// TwinCAT 3 PLC project PShell_SampleTests
// ProgramVersion: 3.1.4023.0
// libraries:
//   CmpBitmapPool, * (System)
//   PShEll Universal Blocks, * (Precision Systems Engineering)
//   Tc2_MC2, * (Beckhoff Automation GmbH)
//   Tc2_Standard, * (Beckhoff Automation GmbH)
//   Tc2_System, * (Beckhoff Automation GmbH)
//   Tc2_TcpIp, * (Beckhoff Automation GmbH)
//   Tc3_EventLogger, * (Beckhoff Automation GmbH)
//   Tc3_McCollisionAvoidance, * (Beckhoff Automation GmbH)
//   Tc3_McCoordinatedMotion, * (Beckhoff Automation GmbH)
//   Tc3_Module, * (Beckhoff Automation GmbH)
//   VisuDialogs, * (System)
//   VisuSymbols,3.5.10.0,System
// project tree:
//   DUTs/Fixture/ E_FcqFixtureStateGSampleMeas.TcDUT, E_FixtureJigStateAbort.TcDUT, E_FixtureJigStateInit.TcDUT, E_FixtureJigStateReset.TcDUT, E_FixtureLoadNormResult.TcDUT, E_FixtureMeasurementResultExt.TcDUT, E_FixtureState.TcDUT, E_FixtureStateAbort.TcDUT, E_FixtureStateInit.TcDUT, E_FixtureStateLoadNorm.TcDUT, E_FixtureStateMeasurement.TcDUT, E_FixtureStateMeasurementDataExchange.TcDUT, E_FixtureStateReset.TcDUT, E_FixtureStateTest.TcDUT, E_GoldenSampleState.TcDUT
//   DUTs/ ST_Shell.TcDUT, ST_ShellFlags.TcDUT, ST_ShellPlatform.TcDUT, ST_ShellRecipeData.TcDUT
//   / GlobalTextList.TcGTLO, RecipeManager.TcRMO (not stored), SampleTests.TcTTO, VisualizationManager.TcVMO (not stored), VISU_TASK.TcTTO
//   GVLs/ GVL.TcGVL
//   POUs/Platform Tests/Alarm Control/ PRG_AlarmControl.TcPOU
//   POUs/Platform Tests/Machine Control/ FB_MachineControl.TcPOU, I_MachineControl.TcIO, PRG_MachineControl.TcPOU
//   POUs/Platform Tests/Visu Control/ FB_VisuControl.TcPOU, F_CloseDialog.TcPOU, F_OpenDialog.TcPOU, PRG_VisuControl.TcPOU
//   POUs/Platform Tests/Recipes Manager/ PRG_RecipesManager.TcPOU
//   POUs/Universal Blocks/Alarms/ PRG_FB_AlarmControler_Test.TcPOU
//   POUs/Universal Blocks/Analog Devices/Analog Input/ PRG_FB_AnalogInput_Test.TcPOU
//   POUs/Universal Blocks/Analog Devices/Analog Output/ PRG_FB_AnalogOutput_Test.TcPOU
//   POUs/Universal Blocks/Axis CA/ PRG_FB_AxisServoCA_PreTest.TcPOU, PRG_FB_AxisServoCA_Test.TcPOU, PRG_FB_MoverCA_Test.TcPOU, PRG_FB_Axis_JennyScienceEthCA_Test.TcPOU
//   POUs/Universal Blocks/Axis/ PRG_FB_Axis_Faulhaber_Test.TcPOU (excluded from build), PRG_FB_Axis_JennyScienceEthSingle_Test.TcPOU (excluded from build), PRG_FB_AxisServo_Test.TcPOU
//   POUs/Universal Blocks/Communication/Backhoff ADS/ PRG_FB_AdsExchanger_Test.TcPOU
//   POUs/Universal Blocks/Communication/TcpIp/ PRG_FB_TcpClient_Test.TcPOU, PRG_FB_TcpServer_Test.TcPOU, PRG_FUN_TcpDataConversion_Test.TcPOU
//   POUs/Universal Blocks/Cylinder/ PRG_FB_SingleCoilCylinder_Test.TcPOU, PRG_FB_DoubleCoilCylinder_Test.TcPOU
//   POUs/Universal Blocks/Digital Devices/Beacon/ PRG_FB_Beacon_Test.TcPOU
//   POUs/Universal Blocks/Digital Devices/Digital Input/ PRG_FB_DigitalInput_Test.TcPOU, PRG_FB_DigitalInputExt_Test.TcPOU
//   POUs/Universal Blocks/Digital Devices/Digital Output/ PRG_FB_DigitalOutput_Test.TcPOU
//   POUs/Universal Blocks/Digital Devices/Lamp/ PRG_FB_Lamp_Test.TcPOU
//   POUs/Universal Blocks/Fixtures/ FB_Fixture222.TcPOU, PRG_FB_FixtureCommTest.TcPOU
//   POUs/Universal Blocks/Fixture/ FB_FixtureClamp.TcPOU, FB_FixtureJig.TcPOU, FB_Fixture.TcPOU, PRG_FB_FcqFixture_Development_Test.TcPOU
//   POUs/Universal Blocks/Robots/ PRG_FB_CR800.TcPOU
//   POUs/Universal Blocks/Utilities/Beckhoff UPS/ PRG_FB_UpsCx20xx_Test.TcPOU, PRG_FB_UpsCx50xx_Test.TcPOU
//   POUs/Universal Blocks/Utilities/CSV Data Exchanger/ PRG_FB_CSVDataExchanger_Test.TcPOU
//   POUs/Universal Blocks/Utilities/File Logger/ PRG_FB_FileLogger_Test.TcPOU
//   POUs/Universal Blocks/Utilities/Recipes Manager/ PRG_FB_RecipesManager_Test.TcPOU
//   POUs/Universal Blocks/Utilities/StringMerge/ PRG_FUN_MergeStringsX_Test.TcPOU
//   POUs/Universal Blocks/Utilities/TXT Data Exchanger/ PRG_FB_TXTDataExchanger_Test.TcPOU
//   POUs/Universal Blocks/Vision/ PRG_FB_Camera_Test.TcPOU
//   POUs/Universal Blocks/XTS/ FB_XtsStation.TcPOU, PRG_XtsControlUnit_Test.TcPOU
//   VISUs/Platform/Pages/ PageAuto.TcVIS, PageInitializing.TcVIS, PageManualOther.TcVIS, PageUninitialized.TcVIS
//   VISUs/Platform/ ShellMainVisu.TcVIS

CONFIGURATION PShell_SampleTests
    RESOURCE PLC ON TwinCAT3
        TASK SampleTests(INTERVAL := T#10ms, PRIORITY := 20);
        TASK VISU_TASK(INTERVAL := T#200000us, PRIORITY := 30);
        PROGRAM PRG_MachineControl WITH SampleTests : PRG_MachineControl;
        PROGRAM PRG_AlarmControl WITH SampleTests : PRG_AlarmControl;
        PROGRAM PRG_RecipesManager WITH SampleTests : PRG_RecipesManager;
        PROGRAM PRG_VisuControl WITH SampleTests : PRG_VisuControl;
        PROGRAM VisuElems_Visu_Prg WITH VISU_TASK : VisuElems.Visu_Prg;
    END_RESOURCE
END_CONFIGURATION

// ---- DUTs/Fixture/E_FcqFixtureStateGSampleMeas.TcDUT

{attribute 'strict'}
TYPE E_FcqFixtureStateGSampleMeas :
(
	FIXTURE_GOLDEN_SAMPLE_CLOSE								:= 0,
	FIXTURE_GOLDEN_SAMPLE_SEND_MEASURE_COMMAND				:= 10,
	FIXTURE_GOLDEN_SAMPLE_WAIT_FOR_RESPONSE 				:= 20,
	FIXTURE_GOLDEN_SAMPLE_OPEN								:= 30,
	FIXTURE_GOLDEN_SAMPLE_MEASUREMENT_DONE					:= 40,
	FIXTURE_GOLDEN_SAMPLE_WAIT_FOR_UTU						:= 50
	
	
);
END_TYPE

// ---- DUTs/Fixture/E_FixtureJigStateAbort.TcDUT
{attribute 'strict'}
TYPE E_FixtureJigStateAbort :
(
	FIXTURE_JIG_ABORT_JIG_PUSHER	:= 0,	(*  *)
	FIXTURE_JIG_ABORT_DONE			:= 10	(*  *)
);
END_TYPE

// ---- DUTs/Fixture/E_FixtureJigStateInit.TcDUT
{attribute 'strict'}
TYPE E_FixtureJigStateInit :
(
	FIXTURE_JIG_INIT_JIG_PUSHER	:= 0,	(*  *)
	FIXTURE_JIG_INIT_DONE		:= 10	(*  *)
);
END_TYPE

// ---- DUTs/Fixture/E_FixtureJigStateReset.TcDUT
{attribute 'strict'}
TYPE E_FixtureJigStateReset :
(
	FIXTURE_JIG_RESET_JIG_PUSHER	:= 10,	(*  *)
	FIXTURE_JIG_RESET_DONE			:= 0	(*  *)
);
END_TYPE

// ---- DUTs/Fixture/E_FixtureLoadNormResult.TcDUT
{attribute 'strict'}
TYPE E_FixtureLoadNormResult :
(
	FIXTURE_NORM_LOAD_UNKNOWN				:= 0,	(*  *)
	FIXTURE_NORM_LOAD_SUCCESS				:= 10,	(*  *)
	FIXTURE_NORM_LOAD_FAIL					:= 20,	(*  *)
	FIXTURE_NORM_LOAD_GOLDEN_SAMPLE_NEEDED 	:= 30	(*	*)
);
END_TYPE

// ---- DUTs/Fixture/E_FixtureMeasurementResultExt.TcDUT
{attribute 'strict'}
TYPE E_FixtureMeasurementResultExt :
(
	FIXTURE_MEASUREMENT_RESULT_NONE			:= 0,
	FIXTURE_MEASUREMENT_RESULT_GOOD			:= 10,
	FIXTURE_MEASUREMENT_RESULT_THD 			:= 20,
	FIXTURE_MEASUREMENT_RESULT_PHASE		:= 30,
	FIXTURE_MEASUREMENT_RESULT_SSPL			:= 40,
	FIXTURE_MEASUREMENT_RESULT_RUBBING		:= 50,
	FIXTURE_MEASUREMENT_RESULT_IMP			:= 60,
	FIXTURE_MEASUREMENT_RESULT_HFA			:= 70,
	FIXTURE_MEASUREMENT_RESULT_SPL			:= 80,
	FIXTURE_MEASUREMENT_RESULT_CONNECT		:= 90,
	FIXTURE_MEASUREMENT_RESULT_REJECT_OTHER	:= 100,
	FIXTURE_MEASUREMENT_RESULT_REWORK		:= 110
);
END_TYPE

// ---- DUTs/Fixture/E_FixtureState.TcDUT
{attribute 'strict'}
TYPE E_FixtureState :
(
	FIXTURE_EXTENSION_IDLE								:= 0,	(*  *)
	FIXTURE_EXTENSION_COVER_ACTIVE	 					:= 10,	(*  *)
	FIXTURE_EXTENSION_COVER_ACTIVE_DONE					:= 20,	(*  *)
	FIXTURE_EXTENSION_COVER_HOME						:= 30,	(*  *)
	FIXTURE_EXTENSION_COVER_HOME_DONE					:= 40,	(*  *)
	FIXTURE_EXTENSION_CLAMP_HOLD						:= 50,	(*  *)
	FIXTURE_EXTENSION_CLAMP_HOLD_DONE					:= 60,	(*  *)
	FIXTURE_EXTENSION_CLAMP_RELEASE						:= 70,	(*  *)
	FIXTURE_EXTENSION_CLAMP_RELEASE_DONE				:= 80,	(*  *)
	FIXTURE_EXTENSION_COVER_ACTIVE_AND_JIG_OPEN			:= 90,	(*  *)
	FIXTURE_EXTENSION_COVER_ACTIVE_AND_JIG_OPEN_DONE 	:= 100,	(*  *)
	FIXTURE_EXTENSION_COVER_HOME_AND_JIG_CLOSE			:= 110,	(*  *)
	FIXTURE_EXTENSION_COVER_HOME_AND_JIG_CLOSE_DONE		:= 120,	(*  *)
	FIXTURE_EXTENSION_LOAD_NORM							:= 130,	(*  *)
	FIXTURE_EXTENSION_LOAD_NORM_DONE					:= 140,	(*  *)
	FIXTURE_EXTENSION_GOLDEN_SAMPLE_MEASURE				:= 150,	(*	*)
	FIXTURE_EXTENSION_GOLDEN_SAMPLE_MEASURE_DONE		:= 160	(*  *)
);
END_TYPE

// ---- DUTs/Fixture/E_FixtureStateAbort.TcDUT
{attribute 'strict'}
TYPE E_FixtureStateAbort :
(
	FIXTURE_ABORT_CLAMP		:= 0,	(*  *)
	FIXTURE_ABORT_COVER		:= 20,	(*  *)
	FIXTURE_ABORT_DONE	:= 10	(*  *)
);
END_TYPE

// ---- DUTs/Fixture/E_FixtureStateInit.TcDUT
{attribute 'strict'}
TYPE E_FixtureStateInit :
(
	FIXTURE_INIT_CLAMP	:= 0,	(*  *)
	FIXTURE_INIT_COVER	:= 20,	(*  *)
	FIXTURE_INIT_DONE	:= 10	(*  *)
);
END_TYPE

// ---- DUTs/Fixture/E_FixtureStateLoadNorm.TcDUT
{attribute 'strict'}
TYPE E_FixtureStateLoadNorm :
(
	FIXTURE_LOADING_NORM_SEND_NORM_DATA 				:= 0,	(*  *)
	FIXTURE_LOADING_NORM_WAIT_FOR_RESPONSE				:= 10,	(*  *)
	FIXTURE_LOADING_NORM_DONE							:= 20,	(*  *)
	FIXTURE_LOADING_NORM_GOLDEN_SAMPLE_TEST 			:= 30,	(*	*)
	FIXTURE_LOADING_NORM_GOLDEN_SAMPLE_WAIT_FOR_END		:= 40	(*	*)
);
END_TYPE

// ---- DUTs/Fixture/E_FixtureStateMeasurement.TcDUT
{attribute 'strict'}
TYPE E_FixtureStateMeasurement :
(
	FIXTURE_MEASUREMENT_START 				:= 0,
	FIXTURE_MEASUREMENT_WAIT_FOR_BUSY 		:= 10,
	FIXTURE_MEASUREMENT_WAIT_FOR_RESPONSE 	:= 20,
	FIXTURE_MEASUREMENT_REMEASUREMENT		:= 30,
	FIXTURE_MEASUREMENT_DONE				:= 40
);
END_TYPE

// ---- DUTs/Fixture/E_FixtureStateMeasurementDataExchange.TcDUT
{attribute 'strict'}
TYPE E_FixtureStateMeasurementDataExchange :
(
	FIXTURE_MEASURE_DATA_EXCHANGING_WAIT_FOR_BUSY 		:= 0,
	FIXTURE_MEASURE_DATA_EXCHANGING_WAIT_FOR_FISNISH 	:= 10,
	FIXTURE_MEASURE_DATA_EXCHANGING_PROCCESS_RESULTS 	:= 20,
	FIXTURE_MEASURE_DATA_EXCHANGING_DONE				:= 30
);
END_TYPE

// ---- DUTs/Fixture/E_FixtureStateReset.TcDUT
{attribute 'strict'}
TYPE E_FixtureStateReset :
(
	FIXTURE_RESET_CLAMP	:= 0,	(*  *)
	FIXTURE_RESET_COVER	:= 10,	(*  *)
	FIXTURE_RESET_DONE	:= 20	(*  *)
);
END_TYPE

// ---- DUTs/Fixture/E_FixtureStateTest.TcDUT
{attribute 'strict'}
TYPE E_FixtureStateTest :
(
	FIXTURE_TEST_WAIT_FOR_COMMAND 			:= 0,	(*  *)
	FIXTURE_TEST_INIT						:= 10,	(*  *)
	FIXTURE_TEST_OPEN						:= 20,	(*  *)
	FIXTURE_TEST_CLOSE						:= 30,	(*  *)
	FIXTURE_TEST_MEASURE					:= 40,	(*  *)
	FIXTURE_TEST_RESET						:= 50,	(*  *)
	FIXTURE_TEST_PLATFORM_HOME				:= 60,	(*  *)
	FIXTURE_TEST_PLATFORM_ACTIVE			:= 70,	(*  *)
	FIXTURE_TEST_PRODUCT_HOLD				:= 80,	(*  *)
	FIXTURE_TEST_PRODUCT_RELEASE			:= 90,	(*  *)
	FIXTURE_TEST_PLATFORM_ACTIVE_AND_OPEN	:= 100,	(*  *)
	FIXTURE_TEST_PLATFORM_HOME_AND_CLOSE	:= 110,	(*  *)
	FIXTURE_TEST_LOAD_NORM					:= 120,	(*  *)
	FIXTURE_TEST_MEASUREMENT				:= 130,	(*  *)
	FIXTURE_START_POS						:= 210,
	FIXTURE_TEST_HOME						:= 220,
	FIXTURE_TEST_ERROR						:= 999,
	FIXTURE_TEST_ABORT						:= -10	(*  *)
);
END_TYPE

// ---- DUTs/Fixture/E_GoldenSampleState.TcDUT
{attribute 'strict'}
TYPE E_GoldenSampleState :
(
	GS_STATUS_UNKNOWN		:= 0,
	GS_STATUS_BCHECKSETUP	:= 10,
	GS_STATUS_NOK			:= 20,
	GS_STATUS_OK			:= 30
);
END_TYPE

// ---- DUTs/ST_Shell.TcDUT
TYPE ST_Shell :
STRUCT
	stPlatform		: ST_ShellPlatform;		(*  *)
	stFlags			: ST_ShellFlags;		(*  *)
	stRecipeData	: ST_ShellRecipeData;	(*  *)
END_STRUCT
END_TYPE

// ---- DUTs/ST_ShellFlags.TcDUT
TYPE ST_ShellFlags :
STRUCT
	bMachineCtrlAssignamentsDone	: BOOL := FALSE;	(*  *)
	bVisuCtrlAssignamentsDone		: BOOL := FALSE;	(*  *)
	bAlarmCtrlAssignamentsDone		: BOOL := FALSE;	(*  *)
	bRecipesCtrlAssignamentsDone	: BOOL := FALSE;	(*  *)
END_STRUCT
END_TYPE

// ---- DUTs/ST_ShellPlatform.TcDUT
TYPE ST_ShellPlatform EXTENDS ST_UniversalPlatform :
STRUCT
	ref_fbMachineControler : REFERENCE TO FB_MachineControl;	(*  *)
	//refFbMachineSafety	: REFERENCE TO FB_MachineSafety;	(*  *)
	ref_fbVisuControler	: REFERENCE TO FB_VisuControl;			(*  *)
END_STRUCT
END_TYPE

// ---- DUTs/ST_ShellRecipeData.TcDUT
TYPE ST_ShellRecipeData :
STRUCT
	(* Add recipe variables here and link them with RecipeManager in Tc3 XAE Shell *)
	rpVar1 : FB_RecipeParameter;
	rpVar2 : FB_RecipeParameter;
	rpVar3 : FB_RecipeParameter;
	rpVar4 : FB_RecipeParameter;
	rpVar5 : FB_RecipeParameter;
	rpVar6 : FB_RecipeParameter;
	rpVar7 : FB_RecipeParameter;
	rpVar8 : FB_RecipeParameter;
	rpVar9 : FB_RecipeParameter;
    rpVar10 : FB_RecipeParameter;
END_STRUCT
END_TYPE

// ---- GVLs/GVL.TcGVL
VAR_GLOBAL
	stShell : ST_Shell;	(* This structure contains references to Shell modules, recipe parameters and auxilary bit flags *)

	(* Measurement FCQ fixtures *)
	sFIXTURE_NAME								: STRING		:= 'Fixture';
	sFIXTURE_HOST								: T_IPv4Addr	:= '192.168.0.';
	sFIXTURE_AMS_NET_ID							: T_AmsNetID	:= '';
	iFIXTURE_PORT								: UINT			:= 400;
	tFIXTURE_TIMEOUT							: TIME			:= DEFAULT_ADS_TIMEOUT;
	bFIXTURE_USE_LOGGER							: BOOL			:= FALSE;
	bFIXTURE_USE_CLIENT							: BOOL			:= TRUE;
	sFIXTURE_LOGGER_NAME						: STRING		:= 'Logger_Fixture_';
	sFIXTURE_FILE_DIR							: STRING		:= 'C:\Fixture_';
END_VAR

// ---- POUs/Platform Tests/Machine Control/I_MachineControl.TcIO
INTERFACE I_MachineControl EXTENDS I_UniversalMachine

PROPERTY Axes : REFERENCE TO ARRAY[0..19] OF FB_AxisServo
GET
END_GET
END_PROPERTY

PROPERTY DoubleCoilCylinders : REFERENCE TO ARRAY[0..9] OF FB_DoubleCoilCylinder
GET
END_GET
END_PROPERTY

PROPERTY Inputs : REFERENCE TO ARRAY[0..19] OF FB_DigitalInput
GET
END_GET
END_PROPERTY

PROPERTY Outputs : REFERENCE TO ARRAY[0..19] OF FB_DigitalOutput
GET
END_GET
END_PROPERTY

PROPERTY Robots : REFERENCE TO ARRAY[0..9] OF  FB_CR800EtherCAT
GET
END_GET
END_PROPERTY

PROPERTY SafeInputs : REFERENCE TO ARRAY[0..19] OF FB_DigitalInput
GET
END_GET
END_PROPERTY

PROPERTY SafeOutputs : REFERENCE TO ARRAY[0..19] OF FB_DigitalOutput
GET
END_GET
END_PROPERTY

PROPERTY SingleCoilCylinders : REFERENCE TO ARRAY[0..9] OF FB_SingleCoilCylinder
GET
END_GET
END_PROPERTY

END_INTERFACE

// ---- POUs/Platform Tests/Machine Control/PRG_MachineControl.TcPOU
PROGRAM PRG_MachineControl
VAR
	bFirstCycle 		: BOOL := TRUE;			(*  *)
	fbMachineControler 	: FB_MachineControl;	(*  *)
	fbFileLogger 		: FB_FileLogger;		(*	*)
END_VAR

IF bFirstCycle THEN
	bFirstCycle := FALSE;
	
	(* Assign machine controler reference to Shell API*)
	stShell.stPlatform.ref_fbMachineControler REF= fbMachineControler;
	
	(* Set assignamnet done bit for visu controler *)
	stShell.stFlags.bMachineCtrlAssignamentsDone := TRUE;
	
	fbMachineLogger.MR_FirstCycle( 	sName		:= 'PSE_Shell_Machine_Logger',
									sFileDir 	:= 'C:\TwinCAT\Projects\Loggers',
									sFileName 	:= 'PSE_Shell_Machine_Logger',
									sAmsNetId 	:= '',
									bAddTimeStamp := FALSE,
									bAddHeader := FALSE);
END_IF

IF NOT fbMachineLogger.Active THEN 
	fbMachineLogger.MR_Init();	
END_IF

fbMachineTime(bEnable := TRUE);
fbMachineControler();
fbMachineLogger();

END_PROGRAM

// ---- POUs/Platform Tests/Machine Control/FB_MachineControl.TcPOU
FUNCTION_BLOCK FB_MachineControl EXTENDS FB_UniversalMachine IMPLEMENTS I_MachineControl
VAR
	iLoop : USINT;	(* for loop auxilary variable *)

	(* --- Sample actuators - from shell template --- DELETE IF NOT NEEDED - *)
	arrDigitalInput		: ARRAY[0..19] OF FB_DigitalInput;			(* Array of sample digital inputs *)
	arrDigitalOutput	: ARRAY[0..19] OF FB_DigitalOutput;			(* Array of sample digital outputs *)
	arrCylinderDc		: ARRAY[0..9] OF FB_DoubleCoilCylinder;		(* Array of sample double coil cylinders *)
	arrCylinderSc		: ARRAY[0..9] OF FB_SingleCoilCylinder;		(* Array of sample single coil cylinders *)
	arrAxis				: ARRAY[0..19] OF FB_AxisServo;				(* Array of sample axis *)
	arrRobot			: ARRAY[0..9] OF FB_CR800EtherCAT;			(* Array of sample robots *)
	
	tonTestDelay	: TON;	(* Delay which allows to see any page changes during tests *)
	(* --- Sample actuators - from shell template --- DELETE IF NOT NEEDED - *)
	
	bStart			: BOOL;
	
	(* CR800 - testing *)
	lrPositionX1 : LREAL := 203.733;
	lrPositionY1 : LREAL := 100.000;
	lrRotation1  : LREAL := 216.699;
	
	lrPositionX2 : LREAL := -13.733;
	lrPositionY2 : LREAL := 8.001;
	lrRotation2  : LREAL := -2.889;
	
	
	bUserDefinedArea1	: BOOL;
	bTryIt1				: BOOL;
	bTryIt2				: BOOL;
END_VAR

IF bFirstCycle THEN
	(* bFirstCycle bit reset by parent *)
	(* --- Assign initial parameters for machine objects ---*)
	(* ---- DELETE IF NOT NEEDED ---- *)
	(* Assign sample digital inputs *)
	FOR iLoop := 0 TO 19 DO
		arrDigitalInput[iLoop].MR_FirstCycle(CONCAT('Digital_Input_',USINT_TO_STRING(iLoop)),CONCAT('EL1008-',USINT_TO_STRING(iLoop/8)),USINT_TO_STRING(iLoop MOD 8));
	END_FOR
	
	(* Assign sample digital outputs *)
	FOR iLoop := 0 TO 19 DO
		arrDigitalOutput[iLoop].MR_FirstCycle(CONCAT('Digital_Output_',USINT_TO_STRING(iLoop)),CONCAT('EL2008-',USINT_TO_STRING(iLoop/8)),USINT_TO_STRING(iLoop MOD 8));
	END_FOR
	
	(* Assign sample cylinders *)
	FOR iLoop := 0 TO 9 DO
		arrCylinderDc[iLoop].MR_FirstCycle(	sName					:= CONCAT('Double_Coil_Cylinder_',USINT_TO_STRING(iLoop)),
											sActiveSensorModuleType :=CONCAT('EL1008-',USINT_TO_STRING(iLoop/4)),
											sActiveSensorPortID 	:= USINT_TO_STRING(iLoop*2),
											sHomeSensorModuleType	:=CONCAT('EL1008-',USINT_TO_STRING(iLoop/4)),
											sHomeSensorPortID		:= USINT_TO_STRING(iLoop*2+1),
											tGoHomeTimeout			:= T#10S,
											tGoActiveTimeout		:= T#10S,
											tDelay 					:= T#1S);
		arrCylinderDc[iLoop].Simulation := TRUE;
		arrCylinderDc[iLoop].ref_poActiveValve.ModuleType := CONCAT('EL2008-',USINT_TO_STRING(iLoop/4));
		arrCylinderDc[iLoop].ref_poActiveValve.PortID := USINT_TO_STRING(iLoop*2);
		arrCylinderDc[iLoop].ref_poHomeValve.ModuleType := CONCAT('EL2008-',USINT_TO_STRING(iLoop/4));
		arrCylinderDc[iLoop].ref_poHomeValve.PortID := USINT_TO_STRING(iLoop*2+1);
	END_FOR
	
	FOR iLoop := 0 TO 9 DO
		arrCylinderSc[iLoop].MR_FirstCycle(	sName				:= CONCAT('Single_Coil_Cylinder_', USINT_TO_STRING(iLoop)),
											sActiveSensorModuleType :=CONCAT('EL1008-',USINT_TO_STRING(iLoop/4)),
											sActiveSensorPortID :=USINT_TO_STRING(iLoop*2),
											sHomeSensorModuleType :=CONCAT('EL1008-',USINT_TO_STRING(iLoop/4)),
											sHomeSensorPortID	:=USINT_TO_STRING(iLoop*2+1),
											tGoHomeTimeout 		:= T#12S,
											tGoActiveTimeout 	:= T#12S,
											tDelay 				:= T#2S);
		arrCylinderSc[iLoop].Simulation := TRUE;
		arrCylinderSc[iLoop].ref_poActiveValve.ModuleType := CONCAT('EL2008-',USINT_TO_STRING(iLoop/8));
		arrCylinderSc[iLoop].ref_poActiveValve.PortID := USINT_TO_STRING(iLoop);
	END_FOR
	
	(* Assign sample axes *)
	FOR iLoop := 0 TO 19 DO
		arrAxis[iLoop].MR_FirstCycle( 	sName 				:= CONCAT('Axis_',USINT_TO_STRING(iLoop)),
										sMeasurementUnits 	:= 'mm',
										bModulo				:= FALSE);
		arrAxis[iLoop].ref_HomeSwitch.ModuleType :=CONCAT('EL1008-',USINT_TO_STRING(iLoop/8));
		arrAxis[iLoop].ref_HomeSwitch.PortID :=USINT_TO_STRING(iLoop MOD 8);			
	END_FOR	
	
	(* Assign sample robots *)
	FOR iLoop := 0 TO 9 DO
		arrRobot[iLoop].MR_FirstCycle(	sName		:= CONCAT('Robot_',USINT_TO_STRING(iLoop)),
										iOverride	:= 100);
	END_FOR
	(* ---- DELETE IF NOT NEEDED ---- *)
END_IF

(* Execute parent implementation *)
SUPER^();

(* --- Cyclic run of internal objects ---*)
(* ---- DELETE IF NOT NEEDED ---- *)
(* Cyclic run of sample inputs *)
FOR iLoop := 0 TO 19 DO
	arrDigitalInput[iLoop]();
END_FOR

(* Cyclic run of sample outputs *)
FOR iLoop := 0 TO 19 DO
	arrDigitalOutput[iLoop]();
END_FOR
	
(* Cyclic run of sample double coil cylinders *)
FOR iLoop := 0 TO 9 DO
	arrCylinderDc[iLoop]();
END_FOR

(* Cyclic run of sample single coil cylinders *)
FOR iLoop := 0 TO 9 DO
	arrCylinderSc[iLoop]();
END_FOR

(* Cyclic run of sample axis *)
FOR iLoop := 0 TO 19 DO
	arrAxis[iLoop]();
END_FOR

(* Cyclic run of sample robots *)
FOR iLoop := 0 TO 9 DO
	arrRobot[iLoop]();
END_FOR

IF bTryIt1 THEN
	arrRobot[0].MR_SendPosition1( lrPositionX1 := lrPositionX1,
								lrPositionY1 := lrPositionY1,
								lrRotation1  := lrRotation1);
	IF NOT arrRobot[0].SendingPosition1 THEN
		bTryIt1 := FALSE;
	END_IF
END_IF

IF bTryIt2 THEN
	arrRobot[0].MR_SendPosition2( lrPositionX2 := lrPositionX2,
								lrPositionY2 := lrPositionY2,
								lrRotation2  := lrRotation2);
	IF NOT arrRobot[0].SendingPosition2 THEN
		bTryIt1 := FALSE;
	END_IF
END_IF

bUserDefinedArea1 := arrRobot[0].UserDefinedArea1;

tonTestDelay();
(* ---- DELETE IF NOT NEEDED ---- *)

PROPERTY Axes : REFERENCE TO ARRAY[0..19] OF FB_AxisServo
GET
Axes REF= arrAxis;
END_GET
END_PROPERTY

PROPERTY DoubleCoilCylinders : REFERENCE TO ARRAY[0..9] OF FB_DoubleCoilCylinder
GET
DoubleCoilCylinders REF= arrCylinderDc;
END_GET
END_PROPERTY

PROPERTY Inputs : REFERENCE TO ARRAY[0..19] OF FB_DigitalInput
GET
Inputs REF= arrDigitalInput;
END_GET
END_PROPERTY

METHOD MR_Start : BOOL
VAR_INPUT
END_VAR
bRunning := TRUE;

IF NOT bStart THEN
	fbMsgAutoStarted.Send(0);
	bStart := TRUE;
END_IF
END_METHOD

METHOD MR_Stop : BOOL
VAR_INPUT
END_VAR
bRunning := FALSE;

IF bStart THEN
	fbMsgAutoStopped.Send(0);
	bStart := FALSE;
END_IF
END_METHOD

METHOD PROTECTED MS_Aborting
VAR_INPUT
END_VAR
(* 
Add here code to abort all machine objects's e.g robots, axes, cylinders. 
At the end add "eMachineState := MACHINE_STATE_UNINITIALIZED;" to finish aborting.
*)
(* Aborting simulation - DELETE *)
tonTestDelay(IN := TRUE, PT:= T#4S);
IF tonTestDelay.Q THEN
	tonTestDelay(IN := FALSE);
	eMachineState := MACHINE_STATE_UNINITIALIZED;
END_IF
END_METHOD

METHOD PROTECTED MS_Auto
VAR_INPUT
END_VAR
(* 
Add here code to perform automatic process.
*)
;
END_METHOD

METHOD PROTECTED MS_AutoToManual
VAR_INPUT
END_VAR
(* 
Add here code to switch machine into manual mode. 
At the end add "eMachineState := MACHINE_STATE_MANUAL;" to finish switching.
*)
(* Switching mode to manual simulation - DELETE *)
tonTestDelay(IN := TRUE, PT:= T#4S);
bRunning := FALSE;
IF tonTestDelay.Q THEN
	tonTestDelay(IN := FALSE);
	eMachineState := MACHINE_STATE_MANUAL;
END_IF
END_METHOD

METHOD PROTECTED MS_Emergency
VAR_INPUT
END_VAR
END_METHOD

METHOD PROTECTED MS_Initializing
VAR_INPUT
END_VAR
(* 
Add here code to initialize all machine objects's e.g robots, axes, cylinders. 
At the end add "eMachineState := MACHINE_STATE_READY_INITIALIZED;" to finish initialization.
*)
(* Initialization simulation - DELETE  *)
tonTestDelay(IN := TRUE, PT:= T#4S);
IF tonTestDelay.Q THEN
	tonTestDelay(IN := FALSE);
	eMachineState := MACHINE_STATE_READY_INITIALIZED;
END_IF
END_METHOD

METHOD PROTECTED MS_Manual
VAR_INPUT
END_VAR
(* 
Leave empty - manual mode is provided by HMI controler and automatic frame generator.
*)
;
END_METHOD

METHOD PROTECTED MS_ManualToAuto
VAR_INPUT
END_VAR
(* 
Add here code to switch machine into auto mode. 
At the end add "eMachineState := MACHINE_STATE_MANUAL;" to finish switching.
*)
(* Switching mode to auto simulation - DELETE *)
tonTestDelay(IN := TRUE, PT:= T#4S);
IF tonTestDelay.Q THEN
	tonTestDelay(IN := FALSE);
	eMachineState := MACHINE_STATE_AUTO;
END_IF
END_METHOD

METHOD PROTECTED MS_ReadyInitialized
VAR_INPUT
END_VAR
(*
Add code here if some internal parameters are needed to set after initialization or leave it default.
At the end add "eMachineState := MACHINE_STATE_AUTO;" to finish and go to IDLE state.
*)
(* Ready-Initialized simulation - DELETE  *)
tonTestDelay(IN := TRUE, PT:= T#4S);
IF tonTestDelay.Q THEN
	tonTestDelay(IN := FALSE);
	eMachineState := MACHINE_STATE_AUTO;
END_IF
END_METHOD

METHOD PROTECTED MS_Reset
VAR_INPUT
END_VAR
(* 
Add here code to reset all machine objects's e.g robots, axes, cylinders. 
At the end add "eMachineState := MACHINE_STATE_RESET_DONE;" to finish reseting.
*)
(* Reset simulation - DELETE  *)
tonTestDelay(IN := TRUE, PT:= T#4S);
IF tonTestDelay.Q THEN
	tonTestDelay(IN := FALSE);
	eMachineState := MACHINE_STATE_RESET_DONE;
END_IF
END_METHOD

METHOD PROTECTED MS_ResetDone
VAR_INPUT
END_VAR
eMachineState := eMachineStateBeforeReset;
END_METHOD

METHOD PROTECTED MS_Uninitialized
VAR_INPUT
END_VAR
;
END_METHOD

PROPERTY Outputs : REFERENCE TO ARRAY[0..19] OF FB_DigitalOutput
GET
Outputs REF= arrDigitalOutput;
END_GET
END_PROPERTY

PROPERTY Robots : REFERENCE TO ARRAY[0..9] OF FB_CR800EtherCAT
GET
Robots REF= arrRobot;
END_GET
END_PROPERTY

PROPERTY SafeInputs : REFERENCE TO ARRAY[0..19] OF FB_DigitalInput
GET
SafeInputs REF= arrDigitalInput;
END_GET
END_PROPERTY

PROPERTY SafeOutputs : REFERENCE TO ARRAY[0..19] OF FB_DigitalOutput
GET
SafeOutputs REF= arrDigitalOutput;
END_GET
END_PROPERTY

PROPERTY SingleCoilCylinders : REFERENCE TO ARRAY[0..9] OF FB_SingleCoilCylinder
GET
SingleCoilCylinders REF= arrCylinderSc;
END_GET
END_PROPERTY

END_FUNCTION_BLOCK

// ---- POUs/Platform Tests/Alarm Control/PRG_AlarmControl.TcPOU
PROGRAM PRG_AlarmControl
VAR CONSTANT
	sDEFAULT_NAME		: STRING := 'Alarm Controler Test';	
	sDEFAULT_FILE_PATH	: STRING := 'C:\TwinCAT\Tests\EventLogger\events.csv';
END_VAR
VAR
	bFirstCycle			: BOOL := TRUE;
	fbAlarmControler 	: FB_AlarmControler;
	
	bInit 				: BOOL;
	bAbort				: BOOL;
END_VAR

IF bFirstCycle THEN
	bFirstCycle := FALSE;
	
	fbAlarmControler.MR_FirstCycle( sName		:= sDEFAULT_NAME,
									sFileName	:= sDEFAULT_FILE_PATH);
									
	(* Assign machine controler reference to Shell API*)
	stShell.stPlatform.ref_fbAlarmControler REF= fbAlarmControler;
	
	(* Set assignamnet done bit for visu controler *)
	stShell.stFlags.bAlarmCtrlAssignamentsDone := TRUE;
END_IF

fbAlarmControler();

END_PROGRAM

// ---- POUs/Platform Tests/Recipes Manager/PRG_RecipesManager.TcPOU
PROGRAM PRG_RecipesManager
VAR CONSTANT
	sDEFAULT_STORAGE_PATH		: STRING(512) := 'C:\TwinCAT\Tests\Recipes\';	(* Default storage path for recipe files *)
	sDEFAULT_RECIPE_DEFINITION	: STRING := 'Recipes';						(* Default definition of Recipe configuration from RecipesManager *)
	sDEFAULT_RECIPE_NAME		: STRING := 'R1';							(* Default name of selected Recipe *)
END_VAR
VAR		
	bFirstCycle 		: BOOL := TRUE;
	sTest1 				: REFERENCE TO STRING;
	fbRecipesControler	: FB_RecipesControler;	(* Recipes Controler *)
END_VAR

IF bFirstCycle AND fbRecipesControler.RecipeValuesAdrAvailable THEN
	bFirstCycle := FALSE;
	fbRecipesControler.MR_FirstCycle(	sLocalStoragePath 	:= sDEFAULT_STORAGE_PATH,
										sRecipesDefinition	:= sDEFAULT_RECIPE_DEFINITION,
										sDefaultRecipeName	:= sDEFAULT_RECIPE_NAME);					
	
	(* Assign recipe parameters *)								
	stShell.stRecipeData.rpVar1.MR_FirstCycle(	eType := VISU_CTRL_RECIPES_PARAMETER_TYPE_REAL, 
												sName := 'Var1', 
												pFileValueAdr := fbRecipesControler.RecipeValuesAdr[0]);
										
	stShell.stRecipeData.rpVar2.MR_FirstCycle(	eType := VISU_CTRL_RECIPES_PARAMETER_TYPE_REAL, 
												sName := 'Var2', 
												pFileValueAdr := fbRecipesControler.RecipeValuesAdr[1]);
												
	stShell.stRecipeData.rpVar3.MR_FirstCycle(	eType := VISU_CTRL_RECIPES_PARAMETER_TYPE_REAL, 
												sName := 'Var3', 
												pFileValueAdr := fbRecipesControler.RecipeValuesAdr[2]);
												
	stShell.stRecipeData.rpVar4.MR_FirstCycle(	eType := VISU_CTRL_RECIPES_PARAMETER_TYPE_INT, 
												sName := 'Var4', 
												pFileValueAdr := fbRecipesControler.RecipeValuesAdr[3]);			
												
	stShell.stRecipeData.rpVar5.MR_FirstCycle(	eType := VISU_CTRL_RECIPES_PARAMETER_TYPE_INT, 
												sName := 'Var5', 
												pFileValueAdr := fbRecipesControler.RecipeValuesAdr[4]);
												
	stShell.stRecipeData.rpVar6.MR_FirstCycle(	eType := VISU_CTRL_RECIPES_PARAMETER_TYPE_INT, 
												sName := 'Var6', 
												pFileValueAdr := fbRecipesControler.RecipeValuesAdr[5]);
												
	stShell.stRecipeData.rpVar7.MR_FirstCycle(	eType := VISU_CTRL_RECIPES_PARAMETER_TYPE_STRING, 
												sName := 'Var7', 
												pFileValueAdr := fbRecipesControler.RecipeValuesAdr[6]);
												
	stShell.stRecipeData.rpVar8.MR_FirstCycle(	eType := VISU_CTRL_RECIPES_PARAMETER_TYPE_STRING, 
												sName := 'Var8', 
												pFileValueAdr := fbRecipesControler.RecipeValuesAdr[7]);
												
	stShell.stRecipeData.rpVar9.MR_FirstCycle(	eType := VISU_CTRL_RECIPES_PARAMETER_TYPE_STRING, 
												sName := 'Var9', 
												pFileValueAdr := fbRecipesControler.RecipeValuesAdr[8]);
												
	stShell.stRecipeData.rpVar10.MR_FirstCycle(	eType := VISU_CTRL_RECIPES_PARAMETER_TYPE_BOOL, 
												sName := 'Var10', 
												pFileValueAdr := fbRecipesControler.RecipeValuesAdr[9]);
	
	(* Assign recipes controler reference to Shell API*)
	stShell.stPlatform.ref_fbRecipesManager REF= fbRecipesControler;
	
	(* Set assignamnet done bit for visu controler *)
	stShell.stFlags.bRecipesCtrlAssignamentsDone := TRUE;
END_IF

fbRecipesControler();

END_PROGRAM

// ---- POUs/Platform Tests/Visu Control/PRG_VisuControl.TcPOU
PROGRAM PRG_VisuControl
VAR
	iLoop 			: USINT;			(*  *)
	bFirstCycle 	: BOOL := TRUE;		(*  *)
	fbVisuControl	: FB_VisuControl;	(*  *)
END_VAR

IF bFirstCycle AND stShell.stFlags.bMachineCtrlAssignamentsDone AND stShell.stFlags.bAlarmCtrlAssignamentsDone AND stShell.stFlags.bRecipesCtrlAssignamentsDone THEN
	bFirstCycle := FALSE;
	
	fbVisuControl.MR_FirstCycle( 	sMachineName 		:= sMACHINE_NAME,
									sSoftwareVersion	:= sSOFTWARE_VERSION);
									
	(*--- Append platform objects to HMI ---*)
	(* Apped machine controler to HMI controler *)
	fbVisuControl.MR_AppendUniversalMachine(ifMachine := stShell.stPlatform.ref_fbMachineControler);
	
	(* Append alarm controler to HMI controler *)
	fbVisuControl.MR_AppendAlarmControler(ifAlarmControler := stShell.stPlatform.ref_fbAlarmControler);
	
	(* Append recipes manager to HMI controler *)
	fbVisuControl.MR_AppendRecipesManager(ifRecipesManager := stShell.stPlatform.ref_fbRecipesManager);
	
	(* --- Append recipes parameters --- *)
	fbVisuControl.MR_AppendRecipeParameter( ifRecipeParameter := stShell.stRecipeData.rpVar1);
	fbVisuControl.MR_AppendRecipeParameter( ifRecipeParameter := stShell.stRecipeData.rpVar2);
	fbVisuControl.MR_AppendRecipeParameter( ifRecipeParameter := stShell.stRecipeData.rpVar3);
	fbVisuControl.MR_AppendRecipeParameter( ifRecipeParameter := stShell.stRecipeData.rpVar4);
	fbVisuControl.MR_AppendRecipeParameter( ifRecipeParameter := stShell.stRecipeData.rpVar5);
	fbVisuControl.MR_AppendRecipeParameter( ifRecipeParameter := stShell.stRecipeData.rpVar6);
	fbVisuControl.MR_AppendRecipeParameter( ifRecipeParameter := stShell.stRecipeData.rpVar7);
	fbVisuControl.MR_AppendRecipeParameter( ifRecipeParameter := stShell.stRecipeData.rpVar8);
	fbVisuControl.MR_AppendRecipeParameter( ifRecipeParameter := stShell.stRecipeData.rpVar9);
	fbVisuControl.MR_AppendRecipeParameter( ifRecipeParameter := stShell.stRecipeData.rpVar10);
	
	(* --- Append machine objects to HMI ---*)
	(* Append sample digital inputs *)
	FOR iLoop := 0 TO 19 DO
		fbVisuControl.MR_AppendInput(ifDigitalInput := stShell.stPlatform.ref_fbMachineControler.Inputs[iLoop]);
	END_FOR
	
	(* Append sample digital outputs *)
	FOR iLoop := 0 TO 19 DO
		fbVisuControl.MR_AppendOutput(ifDigitalOutput := stShell.stPlatform.ref_fbMachineControler.Outputs[iLoop]);
	END_FOR
	
	(* Append sample digital inputs *)
	FOR iLoop := 0 TO 19 DO
		fbVisuControl.MR_AppendSafeInput(ifSafeInput := stShell.stPlatform.ref_fbMachineControler.SafeInputs[iLoop]);
	END_FOR
	
	(* Append sample digital outputs *)
	FOR iLoop := 0 TO 19 DO
		fbVisuControl.MR_AppendSafeOutput(ifSafeOutput := stShell.stPlatform.ref_fbMachineControler.SafeOutputs[iLoop]);
	END_FOR
	
	(* Append sample double coil cylinders *)
	FOR iLoop := 0 TO 9 DO
		fbVisuControl.MR_AppendCylinder( 	ifCylinder 			:= stShell.stPlatform.ref_fbMachineControler.DoubleCoilCylinders[iLoop],
											eCylinderType 		:= CYLINDER_TYPE_DOUBLE_COIL,
											sActiveDescription	:= 'Active',
											sHomeDescription	:= 'Home');
	END_FOR
	
	(* Append sample single coil cylinders *)
	FOR iLoop := 0 TO 9 DO
		fbVisuControl.MR_AppendCylinder( 	ifCylinder 			:= stShell.stPlatform.ref_fbMachineControler.SingleCoilCylinders[iLoop],
											eCylinderType 		:= CYLINDER_TYPE_SINGLE_COIL,
											sActiveDescription 	:= 'Active',
											sHomeDescription 	:= 'Home');
	END_FOR
	(* Append sample scara robot *)
	FOR iLoop := 0 TO 4 DO
		fbVisuControl.MR_AppendRobot(	ifRobot 	:= stShell.stPlatform.ref_fbMachineControler.Robots[iLoop],
										eRobotType	:= ROBOT_TYPE_MITSUBISHI_SCARA);
	END_FOR
	
	(* Append sample 6 axis robot *)
	FOR iLoop := 5 TO 9 DO
		fbVisuControl.MR_AppendRobot(	ifRobot 	:= stShell.stPlatform.ref_fbMachineControler.Robots[iLoop],
										eRobotType	:= ROBOT_TYPE_MITSUBISHI_6_AXIS);
	END_FOR
	
	(* Append sample axes *)
	FOR iLoop := 0 TO 19 DO
		fbVisuControl.MR_AppendAxis(	ifMotor		:= stShell.stPlatform.ref_fbMachineControler.Axes[iLoop],
										eMotorType	:= AXIS_TYPE_BECKHOFF_XTS_MOVER);
	END_FOR

	(* Set assignamnet done bit *)
	stShell.stFlags.bVisuCtrlAssignamentsDone := TRUE;
END_IF

(* Start running Visu Controler if all other controlers are assigned *)
IF stShell.stFlags.bVisuCtrlAssignamentsDone THEN
	fbVisuControl();
END_IF

END_PROGRAM

// ---- POUs/Platform Tests/Visu Control/FB_VisuControl.TcPOU
FUNCTION_BLOCK FB_VisuControl EXTENDS FB_UniversalVisu
VAR
END_VAR

bBackupRestoreDisabled := TRUE;
SUPER^();

METHOD PROTECTED  MS_Emergency
;
END_METHOD

END_FUNCTION_BLOCK

// ---- POUs/Platform Tests/Visu Control/F_CloseDialog.TcPOU
FUNCTION F_CloseDialog : BOOL
VAR_INPUT
	sDialogName : STRING;
END_VAR
VAR
	pstClientData : POINTER TO VisuElems.VisuStructClientData;
	itfDialogManager : VisuElems.IDialogManager;
	itfMyDialog : VisuElems.IVisualisationDialog;
	stVisuRect : VisuElems.VisuStructSimpleRectangle;
END_VAR

VisuElems.VisuElemBase.g_ClientManager.BeginIteration();
pstClientData := VisuElems.VisuElemBase.g_ClientManager.GetNextClient();
WHILE pstClientData <> 0 DO
   IF pstClientData^.GlobalData.ClientType = VisuElems.Visu_ClientType.HMITargetVisualization THEN
      itfDialogManager := VisuElems.g_VisuManager.GetDialogManager();
      itfMyDialog := itfDialogManager.GetDialog(sDialogName);
      itfDialogManager.CloseDialog	(itfMyDialog, pstClientData);
   END_IF
   pstClientData := VisuElems.VisuElemBase.g_ClientManager.GetNextClient();
END_WHILE

END_FUNCTION

// ---- POUs/Platform Tests/Visu Control/F_OpenDialog.TcPOU
FUNCTION F_OpenDialog : BOOL
VAR_INPUT
	sDialogName : STRING;
END_VAR
VAR
	pstClientData : POINTER TO VisuElems.VisuStructClientData;
	itfDialogManager : VisuElems.IDialogManager;
	itfMyDialog : VisuElems.IVisualisationDialog;
	stVisuRect : VisuElems.VisuStructSimpleRectangle;
END_VAR

VisuElems.VisuElemBase.g_ClientManager.BeginIteration();
pstClientData := VisuElems.VisuElemBase.g_ClientManager.GetNextClient();
WHILE pstClientData <> 0 DO
   IF pstClientData^.GlobalData.ClientType = VisuElems.Visu_ClientType.HMITargetVisualization THEN
      itfDialogManager := VisuElems.g_VisuManager.GetDialogManager();
      itfMyDialog := itfDialogManager.GetDialog(sDialogName);
      stVisuRect.ptTopLeft.iX := ANY_TO_INT(INT#0);
      stVisuRect.ptTopLeft.iY := ANY_TO_INT(INT#0);
      stVisuRect.ptBottomRight.iX := ANY_TO_INT(10);
      stVisuRect.ptBottomRight.iY := ANY_TO_INT(10);
      itfDialogManager.OpenDialog(itfMyDialog, pstClientData, FALSE, ADR(stVisuRect));
   END_IF
   pstClientData := VisuElems.VisuElemBase.g_ClientManager.GetNextClient();
END_WHILE

END_FUNCTION

// ---- POUs/Universal Blocks/Alarms/PRG_FB_AlarmControler_Test.TcPOU
PROGRAM PRG_FB_AlarmControler_Test
VAR
	bFirstCycle			: BOOL := TRUE;
	sName				: STRING := 'Alarm Controler Test';	

	(* Function blocks *)
	fbAlarmControler	: FB_AlarmControler;
	fbTestMessage		: FB_TcMessage;
	fbTestAlarm			: FB_TcAlarm;
	fbTestAlarm2		: FB_TcAlarm;
	
	(* Auxilary test commands *)
	bInit 				: BOOL;
	bAbort 				: BOOL;
	bClear				: BOOL;
	bClearAll 			: BOOL;
	bConfirm 			: BOOL;
	bConfirmAll 		: BOOL;
	bExport 			: BOOL;
	
	bRaiseAlarm			: BOOL;
	bAddMessage 		: BOOL;
	bRaiseAlarm2		: BOOL;
	
	(* Auxilary test parameters *)
	bResetConfirmation 	: BOOL := TRUE;
	sFileName			: STRING := 'C:\TwinCAT\Tests\EventLogger\events.csv';
	
	(* Auxilary test status *)
	bActive 			: BOOL;
	bBusy				: BOOL;
	bError				: BOOL;
	iErrorID 			: UDINT;
	eState				: E_AlarmControlerState;
	
	iState : USINT;
	
END_VAR

IF bFirstCycle THEN
	bFirstCycle := FALSE;
	fbAlarmControler.MR_FirstCycle( sName := sName,
									sFileName := sFileName);
									
	//fbTestMessage.CreateEx(TC_EVENTS.TestEventClass.TestMessage,0);
	//fbTestAlarm.CreateEx(TC_EVENTS.TestEventClass.TestAlarm1,TRUE,0);
	//fbTestAlarm2.CreateEx(TC_EVENTS.TestEventClass.TestAlarm2,FALSE,0);
END_IF

IF bAddMessage THEN
	bAddMessage := FALSE;
	fbTestMessage.Send(0);
	
ELSIF bRaiseAlarm THEN
	bRaiseAlarm := FALSE;
	fbTestAlarm.Raise(0);

ELSIF bRaiseAlarm2 THEN
	bRaiseAlarm2 := FALSE;
	fbTestAlarm2.Raise(0);
	
END_IF

bActive := fbAlarmControler.Active;
bBusy := fbAlarmControler.Busy;
bError := fbAlarmControler.Error;
eState := fbAlarmControler.State;

CASE iState OF
	0:
		IF bInit THEN
			bInit := FALSE;
			iState := 10;
			
		ELSIF bAbort THEN
			bAbort := FALSE;
			iState := 20;
			
		ELSIF bClear THEN
			bClear := FALSE;
			iState := 30;
			
		ELSIF bClearAll THEN
			bClearAll := FALSE;
			iState := 40;
			
		ELSIF bConfirm THEN
			bConfirm := FALSE;
			iState := 50;
			
		ELSIF bConfirmAll THEN
			bConfirmAll := FALSE;
			iState := 60;
			
		ELSIF bExport THEN
			bExport := FALSE;
			iState := 70;
			
		END_IF
	10:
		fbAlarmControler.MR_Init();
		
		IF fbAlarmControler.Active THEN
			iState := 0;
		END_IF
	20:
		fbAlarmControler.MR_Abort();
		
		IF NOT fbAlarmControler.Active THEN
			iState := 0;
		END_IF
	30:
		fbAlarmControler.MR_Clear(0,bResetConfirmation);
		
		IF NOT fbAlarmControler.Busy THEN
			iState := 0;
		END_IF
	40:
		fbAlarmControler.MR_ClearAll(bResetConfirmation);
		
		IF NOT fbAlarmControler.Busy THEN
			iState := 0;
		END_IF
	50:
		fbAlarmControler.MR_Confirm(0);
		
		IF NOT fbAlarmControler.Busy THEN
			iState := 0;
		END_IF
	60:
		fbAlarmControler.MR_ConfirmAll(bResetConfirmation);
		
		IF NOT fbAlarmControler.Busy THEN
			iState := 0;
		END_IF
	70:
		fbAlarmControler.MR_Export();
		
		IF NOT fbAlarmControler.Busy THEN
			iState := 0;
		END_IF
		
END_CASE

fbAlarmControler();

END_PROGRAM

// ---- POUs/Universal Blocks/Analog Devices/Analog Input/PRG_FB_AnalogInput_Test.TcPOU
PROGRAM PRG_FB_AnalogInput_Test
VAR
	bFirsCycle		: BOOL := TRUE;		(* First cycle flag *)
	
	rValue			: REAL;				(* Value from object property *)
	rValueForce		: REAL;				(* Value send to force method *)
	bSetForceValue 	: BOOL;				(* Enable forcing  *)
	
	rValueMin 		: REAL := 0.0;		(*  *)
	rValueMax		: REAL := 10.0;		(*  *)
	rChannelMin		: REAL := 0.0;		(*  *)
	rChannelMax		: REAL := 32767.0;	(*  *)
	
	fbAnalogInput 	: FB_AnalogInput;	(* Analog input object *)
END_VAR

(* Set properties *)
IF bFirsCycle THEN
	bFirsCycle := FALSE;
	fbAnalogInput.MR_FirstCycle( 	sName 			:= 'My test analog input',
									rValueScaledMin := rValueMin,
									rValueScaledMax := rValueMax,
									rChannelMin 	:= rChannelMin,
									rChannelMax 	:= rChannelMax);
END_IF

(* Enable to force channel value *)
IF bSetForceValue THEN
	fbAnalogInput.EnableForce := TRUE;
	fbAnalogInput.MR_SetForceValue(rValueForce);
ELSE
	fbAnalogInput.EnableForce := FALSE;
END_IF

(* Scaned value direct from FB *)
rValue := fbAnalogInput.Value;

fbAnalogInput.ChannelMin	:= rChannelMin;
fbAnalogInput.ChannelMax 	:= rChannelMax;
fbAnalogInput.ValueMin 		:= rValueMin;
fbAnalogInput.ValueMax 		:= rValueMax;
fbAnalogInput();

END_PROGRAM

// ---- POUs/Universal Blocks/Analog Devices/Analog Output/PRG_FB_AnalogOutput_Test.TcPOU
PROGRAM PRG_FB_AnalogOutput_Test
VAR
	bFirsCycle		: BOOL := TRUE;		(* First cycle flag *)
	rValue			: REAL;				(* Scaled value that is send to channel *)
	
	rValueMin 		: REAL := 0.0;		(*  *)
	rValueMax		: REAL := 10.0;		(*  *)
	rChannelMin		: REAL := 0.0;		(*  *)
	rChannelMax		: REAL := 32767.0;	(*  *)
	
	fbAnalogOutput	: FB_AnalogOutput;	(* Analog input object *)
END_VAR

(* Set properties *)
IF bFirsCycle THEN
	bFirsCycle := FALSE;
	fbAnalogOutput.MR_FirstCycle( 	sName 			:= 'My test analog output',
									rValueScaledMin := rValueMin,
									rValueScaledMax := rValueMax,
									rChannelMin 	:= rChannelMin,
									rChannelMax		:= rChannelMax);
END_IF

(* Cyclic properties update *)
fbAnalogOutput.ChannelMin	:= rChannelMin;
fbAnalogOutput.ChannelMax 	:= rChannelMax;
fbAnalogOutput.ValueMin 	:= rValueMin;
fbAnalogOutput.ValueMax 	:= rValueMax;

(* Send value to channel *)
fbAnalogOutput.Value 		:= rValue;
fbAnalogOutput();

END_PROGRAM

// ---- POUs/Universal Blocks/Axis CA/PRG_FB_AxisServoCA_PreTest.TcPOU
PROGRAM PRG_FB_AxisServoCA_PreTest
VAR
	bFirstCycle : BOOL := TRUE;
	
	AxesGroupRef		: AXES_GROUP_REF;
	stAxisRef			: AXIS_REF;
	
	fbAxisCA1			: FB_AxisServoCA;
	fbAxisCA2			: FB_AxisServoCA;
	
	fbAddAxisToGroup 	: MC_AddAxisToGroup;
	fbGroupEnable		: MC_GroupEnable;
	fbGroupReset		: MC_GroupReset;
	
	fbReadGroupStatus	: MC_GroupReadStatus;
	fbReadGroupError	: MC_GroupReadError;
	
	fbMcMoveAbsCA 		: MC_MoveAbsoluteCA;
	
	iState : INT;
	
	bAdd		: BOOL;
	bReset		: BOOL;
	bInit 		: BOOL;
	bDeinit 	: BOOL;
	bHome		: BOOL;
	bMoveAbsCA1 : BOOL;
	bMoveAbsCA2 : BOOL;
	bStop 		: BOOL;
	bHalt: BOOL;
	
	rHomePosition 		: REAL := 0.0;
	rTargetPositionCA1 	: REAL;
	rTargetPositionCA2 	: REAL;
	
	bAdded : BOOL;
	
	lrOverride: LREAL;
	lrVelocity: LREAL;
	lrAcceleration: LREAL;
	lrDeceleration: LREAL;
	lrJerk: LREAL;
	lrJogVelocity: LREAL;
	lrJogAcceleration: LREAL;
	lrJogDeceleration: LREAL;
	lrJogJerk: LREAL;
	lrStopDeceleration: LREAL;
	lrStopJerk: LREAL;
END_VAR

IF bFirstCycle THEN
	bFirstCycle := FALSE;
	
	lrOverride 			:= 100.0;
	lrVelocity 			:= 50.0;
	lrAcceleration		:= 150.0;
	lrDeceleration		:= 150.0;
	lrJerk				:= 150.0;
	
	lrJogVelocity 		:= 25.0;
	lrJogAcceleration	:= 250.0;
	lrJogDeceleration	:= 250.0;
	lrJogJerk			:= 250.0;
	
	lrStopDeceleration	:= 250.0;
	lrStopJerk			:= 250.0;
	
	fbAxisCA1.Override 			:= lrOverride;
	fbAxisCA1.Velocity 			:= lrVelocity;
	fbAxisCA1.Acceleration 		:= lrAcceleration;
	fbAxisCA1.Deceleration 		:= lrDeceleration;
	fbAxisCA1.Jerk 				:= lrJerk;
	fbAxisCA1.StopDeceleration 	:= lrStopDeceleration;
	fbAxisCA1.StopJerk			:= lrStopJerk;
	
	fbAxisCA2.Override 			:= lrOverride;
	fbAxisCA2.Velocity 			:= lrVelocity;
	fbAxisCA2.Acceleration 		:= lrAcceleration;
	fbAxisCA2.Deceleration 		:= lrDeceleration;
	fbAxisCA2.Jerk 				:= lrJerk;
	fbAxisCA2.StopDeceleration 	:= lrStopDeceleration;
	fbAxisCA2.StopJerk			:= lrStopJerk;
	
END_IF

IF bStop THEN
	bStop := FALSE;
	iState := 100;
ELSIF bHalt THEN
	bHalt := FALSE;
	iState := 110;
END_IF

fbReadGroupStatus( AxesGroup := AxesGroupRef, Enable := TRUE);
fbReadGroupError( AxesGroup := AxesGroupRef, Enable := TRUE);

CASE iState OF
	0:
		IF bAdd THEN
			bAdded := FALSE;
			bAdd := FALSE;
			iState := 10;
		ELSIF bReset THEN
			bReset := FALSE;
			iState := 5;
			
		ELSIF bInit THEN
			bInit := FALSE;
			iState := 50;
			
		ELSIF bDeinit THEN
			bDeinit := FALSE;
			iState := 60;
			
		ELSIF bHome THEN
			bHome := FALSE;
			iState := 70;
		
		ELSIF bMoveAbsCA1 THEN
			bMoveAbsCA1 := FALSE;
			iState := 80;
			
		ELSIF bMoveAbsCA2 THEN
			bMoveAbsCA2 := FALSE;
			iState := 90;
			
		END_IF
	5:
		fbGroupReset( AxesGroup := AxesGroupRef, Execute := TRUE);
		
		IF fbGroupReset.Done THEN
			fbGroupReset( AxesGroup := AxesGroupRef, Execute := FALSE);
			iState := 0;
		END_IF
		
	10:
		stAxisRef := fbAxisCA1.AxisRef;
		fbAddAxisToGroup( 	AxesGroup := AxesGroupRef,
							Axis := stAxisRef,
							Execute := TRUE,
							IdentInGroup := UDINT_TO_IDENTINGROUP(1));
							
		IF fbAddAxisToGroup.Done THEN
			iState := 20;
		END_IF
		
	20:
		fbAddAxisToGroup( AxesGroup := AxesGroupRef , Axis := stAxisRef, Execute := FALSE);
		
		IF NOT fbAddAxisToGroup.Busy THEN
			iState := 30;
		END_IF
		
	30:
		stAxisRef := fbAxisCA2.AxisRef;
		fbAddAxisToGroup( 	AxesGroup := AxesGroupRef,
							Axis := stAxisRef,
							Execute := TRUE,
							IdentInGroup := UDINT_TO_IDENTINGROUP(2));
							
		IF fbAddAxisToGroup.Done THEN
			iState := 40;
		END_IF
		
	40:
		fbAddAxisToGroup( AxesGroup := AxesGroupRef , Axis := stAxisRef, Execute := FALSE);
		
		IF NOT fbAddAxisToGroup.Busy THEN
			bAdded := TRUE;
			iState := 45;
		END_IF
		
	45:
		
		fbGroupEnable( AxesGroup := AxesGroupRef, Execute := TRUE);
		
		IF fbGroupEnable.Done THEN
			fbGroupEnable( AxesGroup := AxesGroupRef, Execute := FALSE);
			iState := 0;
		END_IF
		
	50:
		fbAxisCA1.MR_Init();
		IF fbAxisCA1.State = E_AxisState.AXIS_READY THEN
			iState := 55;
		END_IF
		
	55:
	
		fbAxisCA2.MR_Init();
		IF fbAxisCA2.State = E_AxisState.AXIS_READY THEN
			iState := 0;
		END_IF
		
	60:
		fbAxisCA1.MR_Deinit();
		fbAxisCA2.MR_Deinit();
		
		IF NOT fbAxisCA1.PowerOn AND NOT fbAxisCA2.PowerOn THEN
			iState := 0;
		END_IF
		
	70:
		fbAxisCA1.MR_Home(0.0);
		
		IF fbAxisCA1.IsHomed THEN
			iState := 75;
		END_IF
		
	75:
		fbAxisCA2.MR_Home(3000.0);
		
		IF fbAxisCA2.IsHomed THEN
			iState := 0;
		END_IF
		
	80:
		fbAxisCA1.MR_MoveAbsolute(rTargetPositionCA1);
		
		IF fbAxisCA1.InPosition THEN
			iState := 0;
		END_IF
		
	90:
		fbAxisCA2.MR_MoveAbsolute(rTargetPositionCA2);
		
		IF fbAxisCA2.InPosition THEN
			iState := 0;
		END_IF
		
	100:
		fbAxisCA1.MR_Stop();
		fbAxisCA2.MR_Stop();

		IF fbAxisCA1.Stopped AND fbAxisCA2.Stopped THEN
			iState := 0;
		END_IF;	
	110:
		fbAxisCA1.MR_Halt();
		fbAxisCA2.MR_Halt();
		
		IF fbAxisCA1.Halted AND fbAxisCA2.Halted THEN
			iState := 0;
		END_IF
		
END_CASE

fbAxisCA1();
fbAxisCA2();

END_PROGRAM

// ---- POUs/Universal Blocks/Axis CA/PRG_FB_AxisServoCA_Test.TcPOU
PROGRAM PRG_FB_AxisServoCA_Test
VAR
	bFirstCycle 		: BOOL := TRUE;
	
	stAxisRef			: AXIS_REF;
	iAxisRemoveID		: UINT;
	
	fbAxesGroupCA		: FB_AxesGroupCA;
	fbAxisCA1			: FB_AxisServoCA;
	fbAxisCA2			: FB_AxisServoCA;
	
	iState 				: INT;
	
	bInit 				: BOOL;
	bGroupInit			: BOOL;
	bGroupDeinit 		: BOOL;
	bAdd				: BOOL;
	bRemove				: BOOL;

	bHome				: BOOL;
	bMoveAbsCA1 		: BOOL;
	bMoveAbsCA2 		: BOOL;
	bStop 				: BOOL;
	bHalt				: BOOL;
	
	rHomePositionCA1 	: REAL := 0.0;
	rHomePositionCA2 	: REAL := 3000.0;
	
	rTargetPositionCA1 	: REAL;
	rTargetPositionCA2 	: REAL;
	
	lrOverride			: LREAL;
	lrVelocity			: LREAL;
	lrAcceleration		: LREAL;
	lrDeceleration		: LREAL;
	lrJerk				: LREAL;
	lrJogVelocity		: LREAL;
	lrJogAcceleration	: LREAL;
	lrJogDeceleration	: LREAL;
	lrJogJerk			: LREAL;
	lrStopDeceleration	: LREAL;
	lrStopJerk			: LREAL;
END_VAR

IF bFirstCycle THEN
	bFirstCycle := FALSE;
	
	
	lrOverride 			:= 100.0;
	lrVelocity 			:= 50.0;
	lrAcceleration		:= 150.0;
	lrDeceleration		:= 150.0;
	lrJerk				:= 150.0;
	
	lrJogVelocity 		:= 25.0;
	lrJogAcceleration	:= 250.0;
	lrJogDeceleration	:= 250.0;
	lrJogJerk			:= 250.0;
	
	lrStopDeceleration	:= 250.0;
	lrStopJerk			:= 250.0;
	
	fbAxesGroupCA.MR_FirstCycle('Axes group CA',lrDeceleration,lrJerk);
	
	fbAxisCA1.Override 			:= lrOverride;
	fbAxisCA1.Velocity 			:= lrVelocity;
	fbAxisCA1.Acceleration 		:= lrAcceleration;
	fbAxisCA1.Deceleration 		:= lrDeceleration;
	fbAxisCA1.Jerk 				:= lrJerk;
	fbAxisCA1.StopDeceleration 	:= lrStopDeceleration;
	fbAxisCA1.StopJerk			:= lrStopJerk;
	
	fbAxisCA2.Override 			:= lrOverride;
	fbAxisCA2.Velocity 			:= lrVelocity;
	fbAxisCA2.Acceleration 		:= lrAcceleration;
	fbAxisCA2.Deceleration 		:= lrDeceleration;
	fbAxisCA2.Jerk 				:= lrJerk;
	fbAxisCA2.StopDeceleration 	:= lrStopDeceleration;
	fbAxisCA2.StopJerk			:= lrStopJerk;
	
END_IF
IF fbAxesGroupCA.Error OR fbAxisCA1.Error OR fbAxisCA2.Error THEN
	bGroupInit := FALSE;
	bGroupDeinit := FALSE;
	bMoveAbsCA1 := FALSE;
	bMoveAbsCA2 := FALSE;
	bHome := FALSE;
	bRemove := FALSE;
	iState := 0;
END_IF

IF bStop THEN
	bStop := FALSE;
	iState := 255;
ELSIF bHalt THEN
	bHalt := FALSE;
	iState := 254;
END_IF

CASE iState OF
	0:	
		IF bInit THEN
			bInit := FALSE;
			iState := 10;
			
			
		ELSIF bGroupInit THEN
			bGroupInit := FALSE;
			iState := 50;
			
		ELSIF bGroupDeinit THEN
			bGroupDeinit := FALSE;
			iState := 80;
			
		ELSIF bHome THEN
			bHome := FALSE;
			iState := 90;
		
		ELSIF bMoveAbsCA1 THEN
			bMoveAbsCA1 := FALSE;
			iState := 110;
			
		ELSIF bMoveAbsCA2 THEN
			bMoveAbsCA2 := FALSE;
			iState := 120;
			
		ELSIF bRemove THEN
			bRemove := FALSE;
			iState := 130;
			
		END_IF
	10:
		fbAxisCA1.MR_Init();
		
		IF fbAxisCA1.PowerOn THEN
			iState := 20;
		END_IF
		
	20:
		fbAxisCA2.MR_Init();
		
		IF fbAxisCA2.PowerOn THEN
			iState := 30;
		END_IF
		
	30:
		fbAxisCA1.MR_Home(0.0);
		
		IF fbAxisCA1.IsHomed THEN
			iState := 40;
		END_IF
	40:
		fbAxisCA2.MR_Home(3000.0);
		
		IF fbAxisCA2.IsHomed THEN
			iState := 50;
		END_IF
	50:
		fbAxesGroupCA.MR_Init();
		
		IF fbAxesGroupCA.Active THEN
			iState := 60;
		END_IF
		
	60:
		stAxisRef := fbAxisCA1.AxisRef;
		fbAxesGroupCA.MR_Add(stAxisRef,1);
		
		IF fbAxesGroupCA.AxisAdded THEN
			iState := 70;
		END_IF
		
	70:
		stAxisRef := fbAxisCA2.AxisRef;
		fbAxesGroupCA.MR_Add(stAxisRef,2);
		
		IF fbAxesGroupCA.AxisAdded THEN
			iState := 0;
		END_IF
	80:
		fbAxesGroupCA.MR_Abort();
		
		IF NOT fbAxesGroupCA.Active THEN
			iState := 0;
		END_IF
	90:	
		fbAxisCA1.MR_Home(rHomePositionCA1);
		
		IF fbAxisCA1.IsHomed THEN
			iState := 100;
		END_IF
	100:
		fbAxisCA2.MR_Home(rHomePositionCA2);
		
		IF fbAxisCA2.IsHomed THEN
			iState := 0;
		END_IF
		
	110:
		fbAxisCA1.MR_MoveAbsolute(rTargetPositionCA1);
		
		IF fbAxisCA1.InPosition THEN
			iState := 0;
		END_IF
	120:
		fbAxisCA2.MR_MoveAbsolute(rTargetPositionCA2);
		
		IF fbAxisCA2.InPosition THEN
			iState := 0;
		END_IF
		
	130:
		fbAxesGroupCA.MR_Remove(iAxisRemoveID);
		
		IF fbAxesGroupCA.AxisRemoved THEN
			iState := 0;
		END_IF
		
	254:
		fbAxisCA1.MR_Halt();
		fbAxisCA2.MR_Halt();
		
		IF fbAxisCA1.Halted AND fbAxisCA2.Halted THEN
			iState := 0;
		END_IF
	255:
		fbAxisCA1.MR_Stop();
		fbAxisCA2.MR_Stop();
		
		IF fbAxisCA1.Stopped AND fbAxisCA2.Stopped THEN
			iState := 0;
		END_IF
END_CASE

fbAxisCA1();
fbAxisCA2();
fbAxesGroupCA();

END_PROGRAM

// ---- POUs/Universal Blocks/Axis CA/PRG_FB_MoverCA_Test.TcPOU
PROGRAM PRG_FB_MoverCA_Test
VAR
	bFirstCycle 		: BOOL := TRUE;
	
	stAxisRef			: AXIS_REF;
	iAxisRemoveID		: UINT;
	
	fbAxesGroupCA		: FB_AxesGroupCA;
	fbAxisCA1			: FB_XtsMover;
	fbAxisCA2			: FB_XtsMover;
	
	iState 				: INT;
	
	bInit 				: BOOL;
	bGroupInit			: BOOL;
	bGroupAbort 		: BOOL;
	bAdd				: BOOL;
	bRemove				: BOOL;

	bMoveAbsCA1 		: BOOL;
	bMoveAbsCA2 		: BOOL;
	bStop 				: BOOL;
	bHalt				: BOOL;
	bHaltCA				: BOOL;
	
	lrTargetPositionCA1	: LREAL;
	lrTargetPositionCA2	: LREAL;
	
	lrDistanceCA1		: LREAL;
	lrDistanceCA2		: LREAL;
	
	lrOverride			: LREAL;
	lrVelocity			: LREAL;
	lrAcceleration		: LREAL;
	lrDeceleration		: LREAL;
	lrJerk				: LREAL;
	lrJogVelocity		: LREAL;
	lrJogAcceleration	: LREAL;
	lrJogDeceleration	: LREAL;
	lrJogJerk			: LREAL;
	lrStopDeceleration	: LREAL;
	lrStopJerk			: LREAL;
END_VAR

IF bFirstCycle THEN
	bFirstCycle := FALSE;

	
	lrOverride 			:= 100.0;
	lrVelocity 			:= 100.0;
	lrAcceleration		:= 1000.0;
	lrDeceleration		:= 1000.0;
	lrJerk				:= 10000.0;
	
	lrJogVelocity 		:= 50.0;
	lrJogAcceleration	:= 1000.0;
	lrJogDeceleration	:= 1000.0;
	lrJogJerk			:= 10000.0;
	
	lrStopDeceleration	:= 1000.0;
	lrStopJerk			:= 1000.0;
	
	fbAxesGroupCA.MR_FirstCycle('Axes group CA',lrDeceleration, lrJerk);
	
	fbAxisCA1.Override 			:= lrOverride;
	fbAxisCA1.Velocity 			:= lrVelocity;
	fbAxisCA1.Acceleration 		:= lrAcceleration;
	fbAxisCA1.Deceleration 		:= lrDeceleration;
	fbAxisCA1.Jerk 				:= lrJerk;
	fbAxisCA1.StopDeceleration 	:= lrStopDeceleration;
	fbAxisCA1.StopJerk			:= lrStopJerk;
	
	fbAxisCA2.Override 			:= lrOverride;
	fbAxisCA2.Velocity 			:= lrVelocity;
	fbAxisCA2.Acceleration 		:= lrAcceleration;
	fbAxisCA2.Deceleration 		:= lrDeceleration;
	fbAxisCA2.Jerk 				:= lrJerk;
	fbAxisCA2.StopDeceleration 	:= lrStopDeceleration;
	fbAxisCA2.StopJerk			:= lrStopJerk;
	
END_IF

IF bStop THEN
	bStop := FALSE;
	iState := 255;
ELSIF bHalt THEN
	bHalt := FALSE;
	iState := 254;
END_IF

CASE iState OF
	0:	
		IF bInit THEN
			bInit := FALSE;
			iState := 10;
			
		ELSIF bGroupInit THEN
			bGroupInit := FALSE;
			iState := 30;
			
		ELSIF bGroupAbort THEN
			bGroupAbort := FALSE;
			iState := 60;
		
		ELSIF bMoveAbsCA1 THEN
			bMoveAbsCA1 := FALSE;
			iState := 110;
			
		ELSIF bMoveAbsCA2 THEN
			bMoveAbsCA2 := FALSE;
			iState := 120;
			
		ELSIF bRemove THEN
			bRemove := FALSE;
			iState := 130;
			
		END_IF
	10:
		fbAxisCA1.MR_Init();
		
		IF fbAxisCA1.PowerOn THEN
			iState := 15;
		END_IF
		
	15:
		fbAxisCA1.MR_MoveAbsolute( lrAbsolutePosition := 2000.0);
		
		IF fbAxisCA1.InPosition THEN
			iState := 20;
		END_IF
		
	20:
		fbAxisCA2.MR_Init();
		
		IF fbAxisCA2.PowerOn THEN
			iState := 25;
		END_IF
	
	25:
		fbAxisCA2.MR_MoveAbsolute( lrAbsolutePosition := 1000.0);
		
		IF FBAxisCA2.InPosition THEN
			iState := 0;
		END_IF
	30:
		fbAxesGroupCA.MR_Init();
		
		IF fbAxesGroupCA.Active THEN
			iState := 40;
		END_IF
		
	40:
		stAxisRef := fbAxisCA1.AxisRef;
		fbAxesGroupCA.MR_Add(stAxisRef,1);
		
		IF fbAxesGroupCA.AxisAdded THEN
			iState := 50;
		END_IF
		
	50:
		stAxisRef := fbAxisCA2.AxisRef;
		fbAxesGroupCA.MR_Add(stAxisRef,2);
		
		IF fbAxesGroupCA.AxisAdded THEN
			iState := 0;
		END_IF
		
	60:
		fbAxesGroupCA.MR_Abort();
		
		IF NOT fbAxesGroupCA.Active THEN
			iState := 0;
		END_IF
		
	110:
		fbAxisCA1.Gap := 150.0;
		fbAxisCA1.MR_MoveAbsoluteCA(lrAbsolutePosition := lrTargetPositionCA1);
		
		IF fbAxisCA1.InPosition THEN
			iState := 0;
		END_IF
	120:
		fbAxisCA2.Gap := 150.0;
		fbAxisCA2.MR_MoveAbsoluteCA(lrAbsolutePosition := lrTargetPositionCA2);
		
		IF fbAxisCA2.InPosition THEN
			iState := 0;
		END_IF
		
	130:
		fbAxesGroupCA.MR_Remove(iAxisRemoveID);
		
		IF fbAxesGroupCA.AxisRemoved THEN
			iState := 0;
		END_IF
		
	140:
		fbAxisCA1.MR_MoveRelativeCA( lrRelativeDistance := lrDistanceCA1);
		
		IF fbAxisCA1.InPosition THEN
			iState := 0;
		END_IF
		
	150:
		fbAxisCA2.MR_MoveRelativeCA( lrRelativeDistance := lrDistanceCA2);
		
		IF fbAxisCA2.InPosition THEN
			iState := 0;
		END_IF
	254:
		fbAxisCA1.MR_Halt();
		fbAxisCA2.MR_Halt();
		
		IF fbAxisCA1.Halted AND fbAxisCA2.Halted THEN
			iState := 0;
		END_IF
	255:
		fbAxisCA1.MR_Stop();
		fbAxisCA2.MR_Stop();
		
		IF fbAxisCA1.Stopped AND fbAxisCA2.Stopped THEN
			iState := 0;
		END_IF
END_CASE

fbAxisCA1();
fbAxisCA2();
fbAxesGroupCA();

END_PROGRAM

// ---- POUs/Universal Blocks/Axis CA/PRG_FB_Axis_JennyScienceEthCA_Test.TcPOU
PROGRAM PRG_FB_Axis_JennyScienceEthCA_Test
VAR
	bFirstCycle 		: BOOL := TRUE;
	
	stAxisRef			: AXIS_REF;
	iAxisRemoveID		: UINT;
	
	fbAxesGroupCA		: FB_AxesGroupCA;
	fbAxisCA1			: FB_AxisJennyScienceEthercatCA;
	fbAxisCA2			: FB_AxisJennyScienceEthercatCA;
	
	iState 				: INT;
	
	bInit 				: BOOL;
	bGroupInit			: BOOL;
	bGroupDeinit 		: BOOL;
	bAdd				: BOOL;
	bRemove				: BOOL;

	bHome				: BOOL;
	bMoveAbsCA1 		: BOOL;
	bMoveAbsCA2 		: BOOL;
	bStop 				: BOOL;
	bHalt				: BOOL;
	
	rHomePositionCA1 	: REAL := 0.0;
	rHomePositionCA2 	: REAL := 3000.0;
	
	rTargetPositionCA1 	: REAL;
	rTargetPositionCA2 	: REAL;
	
	lrOverride			: LREAL;
	lrVelocity			: LREAL;
	lrAcceleration		: LREAL;
	lrDeceleration		: LREAL;
	lrJerk				: LREAL;
	lrJogVelocity		: LREAL;
	lrJogAcceleration	: LREAL;
	lrJogDeceleration	: LREAL;
	lrJogJerk			: LREAL;
	lrStopDeceleration	: LREAL;
	lrStopJerk			: LREAL;
END_VAR

IF bFirstCycle THEN
	bFirstCycle := FALSE;
	
	lrOverride 			:= 100.0;
	lrVelocity 			:= 50.0;
	lrAcceleration		:= 150.0;
	lrDeceleration		:= 150.0;
	lrJerk				:= 150.0;
	
	lrJogVelocity 				:= 25.0;
	lrJogAcceleration			:= 250.0;
	lrJogDeceleration			:= 250.0;
	lrJogJerk					:= 250.0;
	
	lrStopDeceleration			:= 250.0;
	lrStopJerk					:= 250.0;
	
	fbAxisCA1.Override 			:= lrOverride;
	fbAxisCA1.Velocity 			:= lrVelocity;
	fbAxisCA1.Acceleration 		:= lrAcceleration;
	fbAxisCA1.Deceleration 		:= lrDeceleration;
	fbAxisCA1.Jerk 				:= lrJerk;
	fbAxisCA1.StopDeceleration 	:= lrStopDeceleration;
	fbAxisCA1.StopJerk			:= lrStopJerk;
	
	fbAxisCA2.Override 			:= lrOverride;
	fbAxisCA2.Velocity 			:= lrVelocity;
	fbAxisCA2.Acceleration 		:= lrAcceleration;
	fbAxisCA2.Deceleration 		:= lrDeceleration;
	fbAxisCA2.Jerk 				:= lrJerk;
	fbAxisCA2.StopDeceleration 	:= lrStopDeceleration;
	fbAxisCA2.StopJerk			:= lrStopJerk;
	
END_IF

IF bStop THEN
	bStop := FALSE;
	iState := 100;
	
ELSIF bHalt THEN
	bHalt := FALSE;
	iState := 110;
	
END_IF

CASE iState OF
	0:	
		IF bInit THEN
			bInit := FALSE;
			iState := 10;
			
			
		ELSIF bGroupInit THEN
			bGroupInit := FALSE;
			iState := 50;
			
		ELSIF bGroupDeinit THEN
			bGroupDeinit := FALSE;
			iState := 80;
			
		ELSIF bHome THEN
			bHome := FALSE;
			iState := 90;
		
		ELSIF bMoveAbsCA1 THEN
			bMoveAbsCA1 := FALSE;
			iState := 110;
			
		ELSIF bMoveAbsCA2 THEN
			bMoveAbsCA2 := FALSE;
			iState := 120;
			
		ELSIF bRemove THEN
			bRemove := FALSE;
			iState := 130;
			
		END_IF
	10:
		fbAxisCA1.MR_Init();
		
		IF fbAxisCA1.PowerOn THEN
			iState := 20;
		END_IF
		
	20:
		fbAxisCA2.MR_Init();
		
		IF fbAxisCA2.PowerOn THEN
			iState := 30;
		END_IF
		
	30:
		fbAxisCA1.MR_Home(0.0);
		
		IF fbAxisCA1.IsHomed THEN
			iState := 40;
		END_IF
	40:
		fbAxisCA2.MR_Home(3000.0);
		
		IF fbAxisCA2.IsHomed THEN
			iState := 50;
		END_IF
	50:
		fbAxesGroupCA.MR_Init();
		
		IF fbAxesGroupCA.Active THEN
			iState := 60;
		END_IF
		
	60:
		stAxisRef := fbAxisCA1.AxisRef;
		fbAxesGroupCA.MR_Add(stAxisRef,1);
		
		IF fbAxesGroupCA.AxisAdded THEN
			iState := 70;
		END_IF
		
	70:
		stAxisRef := fbAxisCA2.AxisRef;
		fbAxesGroupCA.MR_Add(stAxisRef,2);
		
		IF fbAxesGroupCA.AxisAdded THEN
			iState := 0;
		END_IF
	80:
		fbAxesGroupCA.MR_Abort();
		
		IF NOT fbAxesGroupCA.Active THEN
			iState := 0;
		END_IF
	90:	
		fbAxisCA1.MR_Home(rHomePositionCA1);
		
		IF fbAxisCA1.IsHomed THEN
			iState := 100;
		END_IF
	100:
		fbAxisCA2.MR_Home(rHomePositionCA2);
		
		IF fbAxisCA2.IsHomed THEN
			iState := 0;
		END_IF
		
	110:
		fbAxisCA1.MR_MoveAbsolute(rTargetPositionCA1);
		
		IF fbAxisCA1.InPosition THEN
			iState := 0;
		END_IF
	120:
		fbAxisCA2.MR_MoveAbsolute(rTargetPositionCA2);
		
		IF fbAxisCA2.InPosition THEN
			iState := 0;
		END_IF
		
	130:
		fbAxesGroupCA.MR_Remove(iAxisRemoveID);
		
		IF fbAxesGroupCA.AxisRemoved THEN
			iState := 0;
		END_IF
		
	254:
		fbAxisCA1.MR_Halt();
		fbAxisCA2.MR_Halt();
		
		IF fbAxisCA1.Halted AND fbAxisCA2.Halted THEN
			iState := 0;
		END_IF
	255:
		fbAxisCA1.MR_Stop();
		fbAxisCA2.MR_Stop();
		
		IF fbAxisCA1.Stopped AND fbAxisCA2.Stopped THEN
			iState := 0;
		END_IF
END_CASE

fbAxisCA1();
fbAxisCA2();
fbAxesGroupCA();

END_PROGRAM

// ---- POUs/Universal Blocks/Axis/PRG_FB_Axis_Faulhaber_Test.TcPOU
PROGRAM PRG_FB_Axis_Faulhaber_Test
VAR
	bFirstCycle 			: BOOL := TRUE;
	
	bInit					: BOOL;								(* Power on axis and prepare to work *)
	bDeinit					: BOOL;								(* Power off axis and reset status flags *)
	bHome					: BOOL;								(* Home to reference point *)
	bMoveVelocity			: BOOL;								(* Start motion with constant velocity *)
	bMoveAbsolute			: BOOL;								(* Move to absolute position *)
	bMoveAdditive			: BOOL;								(* Move by distance *)
	bMoveRelative			: BOOL;								(* Move by distance *)
	bJog					: BOOL;								(* Start manual jog movement *)
	bStop					: BOOL;								(* High priority stop command *)
	bHalt					: BOOL;								(* Halt current motion, next motion command will abort this command *)
	bReset					: BOOL;								(* Reset axis and return to READY state *)
	
	(* General parameters *)
	bModulo					: BOOL := FALSE;					(* Axis is periodic *)
	lrOverride				: LREAL;							(* Axis velocity override in percents [%] *)
	lrVelocity 				: LREAL;							(* Axis velocirt in measurement units per second *)
	lrAcceleration			: LREAL;							(* Axis acceleration in measurement units per sercond^2 *)
	lrDeceleration 			: LREAL;							(* Axis deceleration in measurement units per sercond^2 *)
	lrJerk					: LREAL;							(* Axis jerk in measurement unit per sercond^3 *)
	lrAbsolutePosition		: LREAL;							(* Target position for MC_MoveAbsolute function *)
	lrRelativeDistance		: LREAL;							(* Relative distance to move for MC_MoveRelative/Additive fuctions *)
	lrHomePosition			: LREAL;							(* This parameters is used to set axis position while performing homing procedure *)
	
	(* Jog function parameters *)	
	lrJogPosition			: LREAL;							(* Relative position to move for jog feature *)
	lrJogVelocity			: LREAL;							(* Jog movement velocity *)
	lrJogAcceleration		: LREAL;							(* Jog movement acceleration *)
	lrJogDeceleration		: LREAL;							(* Jog movement deceleration *)
	lrJogJerk				: LREAL;							(* Jog movement jerk *)
	eJogMode				: E_JogMode;						(* Jog momement mode *)
	eJogDirection			: E_AxisJogDirection;				(* Direction of jog movement *)
	
	(* Stop function parameters *)
	lrStopDeceleration		: LREAL;							(* Stop deceleration *)
	lrStopJerk 				: LREAL;							(* Stop jerk *)
	
	(* Other parameters *)
	stOptions				: ST_MoveOptions;					(* Additional movement options *)
	eDirection				: Tc2_MC2.MC_Direction;				(* Axis movement direction for MC_MoveVelocity *)
	eBufferMode 			: MC_BufferMode := MC_Aborting;		(* Axis buffering mode *)
	
	(* Axis status flags *)
	bActive					: BOOL;
	bBusy					: BOOL;								(* Function block currently executes one of the requests *)
	bError					: BOOL;								(* Error status flag *)
	iErrorID				: UDINT;							(* Error ID *)
	iAxisErrorID			: UDINT;							(* Axis error ID*)
	lrActualPosition		: LREAL;							(* Actual axis position in selected units *)
	rActualVelocity			: REAL;								(* Actual axis velocity in selected units *)
	bPowerOn 				: BOOL;								(* Power On status bit *)
	bIsHomed				: BOOL;								(* Axis has been homed even once *)
	bInVelocity				: BOOL;								(* Axis is moving in target velocity *)
	bInPostion				: BOOL;								(* Axis reached target position *)
	bMoveActive				: BOOL;								(* Axis is moving to target position *)
	bJogDone				: BOOL;								(* Axis manual movement by jog done *)
	bStopped				: BOOL;								(* Axis movement has been stopped *)
	bHalted					: BOOL;								(* Axis movement has been halted *)
	eStatePlcOpen			: E_AxisStatePlcOpen;				(* Current PLCOpen state of axis *)
	
	fbAxis					: FB_AxisFaulhaberLinearMotor;
END_VAR

IF bFirstCycle THEN
	bFirstCycle := FALSE;
	fbAxis.MR_FirstCycle('Faulhaber Linear Motor LM1247 Picker 1 Unit 6','mm', bModulo); //RMA Added bModulo
	
	lrOverride 			:= 100.0;
	lrVelocity 			:= 100.0;
	lrAcceleration		:= 250.0;
	lrDeceleration		:= 250.0;
	lrJerk				:= 250.0;
	lrAbsolutePosition	:= 0.0;
	lrRelativeDistance	:= 0.0;
	lrHomePosition		:= 0.0;
	
	lrJogPosition		:= 0.0;
	lrJogVelocity 		:= 25.0;
	lrJogAcceleration	:= 250.0;
	lrJogDeceleration	:= 250.0;
	lrJogJerk			:= 250.0;
	
	lrStopDeceleration	:= 250.0;
	lrStopJerk			:= 250.0;
	
END_IF

bActive 			:= fbAxis.Active;
bBusy				:= fbAxis.Busy;
bError 				:= fbAxis.Error;
iErrorID 			:= fbAxis.ErrorID;
iAxisErrorID 		:= fbAxis.ErrorID;
lrActualPosition 	:= fbAxis.ActualPosition;
rActualVelocity		:= fbAxis.ActualVelocity;
bPowerOn 			:= fbAxis.PowerOn;
bIsHomed 			:= fbAxis.IsHomed;
bInVelocity			:= fbAxis.InVelocity;
bInPostion 			:= fbAxis.InPosition;
bMoveActive 		:= fbAxis.MoveActive;
bJogDone 			:= fbAxis.JogDone;
bStopped 			:= fbAxis.Stopped;
bHalted 			:= fbAxis.Halted;
eStatePlcOpen		:= fbAxis.StatePlcOpen;

IF bReset THEN
	IF fbAxis.MR_Reset() THEN
		bReset := FALSE;
	END_IF
END_IF

(* Stop commands *)
IF bStop THEN
	bJog := FALSE;
	bMoveAbsolute := FALSE;
	bMoveAdditive := FALSE;
	bMoveRelative := FALSE;
	bMoveVelocity := FALSE;
	
	IF fbAxis.MR_Stop() THEN
		bStop := FALSE;
	END_IF
	
ELSIF bHalt THEN
	bJog := FALSE;
	bMoveAbsolute := FALSE;
	bMoveAdditive := FALSE;
	bMoveRelative := FALSE;
	bMoveVelocity := FALSE;
	
	fbAxis.MR_Halt();
	IF fbAxis.Halted THEN
		bHalt := FALSE;
	END_IF
	
END_IF

(* Other commands *)
IF bInit THEN	
	fbAxis.MR_Init();	
	IF fbAxis.PowerOn THEN
		bInit := FALSE;
	END_IF
	
ELSIF bDeinit THEN
	fbAxis.MR_Abort();
	IF NOT fbAxis.PowerOn THEN
		bDeinit := FALSE;
	END_IF
	
ELSIF bHome THEN
	fbAxis.MR_Home(lrHomePosition);
	IF fbAxis.IsHomed THEN
		bHome := FALSE;
	END_IF
	
ELSIF bMoveVelocity THEN
	fbAxis.MR_MoveVelocity();
	IF fbAxis.InVelocity THEN
		bMoveVelocity := FALSE;
	END_IF
	
ELSIF bMoveAbsolute THEN
	fbAxis.MR_MoveAbsolute(lrAbsolutePosition);
	IF fbAxis.InPosition THEN
		bMoveAbsolute := FALSE;
	END_IF

ELSIF bMoveAdditive THEN
	fbAxis.MR_MoveAdditive(lrRelativeDistance);
	IF fbAxis.InPosition THEN
		bMoveAdditive := FALSE;
	END_IF
	
ELSIF bMoveRelative THEN
	fbAxis.MR_MoveRelative(lrRelativeDistance);
	IF fbAxis.InPosition THEN
		bMoveRelative := FALSE;
	END_IF
	
ELSIF bJog THEN
(*	fbAxis.MR_Jog(lrJogPosition,eJogDirection);
	IF fbAxis.JogDone THEN
		bJog := FALSE;	
	END_IF*)
	
	fbAxis.MR_Jog(bJog); //RMA New jog  
	bJog := FALSE;		//RMA
	
END_IF

fbAxis.Override			:= lrOverride;
fbAxis.Velocity 		:= lrVelocity;
fbAxis.Acceleration 	:= lrAcceleration;
fbAxis.Deceleration 	:= lrDeceleration;
fbAxis.Jerk 			:= lrJerk;
fbAxis.JogVelocity 		:= lrJogVelocity;
fbAxis.JogAcceleration 	:= lrJogAcceleration;
fbAxis.JogDeceleration 	:= lrJogDeceleration;
fbAxis.JogJerk 			:= lrJogJerk;
fbAxis.StopDeceleration := lrStopDeceleration;
fbAxis.StopJerk 		:= lrStopJerk;
	
fbAxis();

END_PROGRAM

// ---- POUs/Universal Blocks/Axis/PRG_FB_Axis_JennyScienceEthSingle_Test.TcPOU
PROGRAM PRG_FB_Axis_JennyScienceEthSingle_Test
VAR
	bFirstCycle 	: BOOL := TRUE;
	
	bInit					: BOOL;								(* Power on axis and prepare to work *)
	bDeinit					: BOOL;								(* Power off axis and reset status flags *)
	bHome					: BOOL;								(* Home to reference point *)
	bMoveVelocity			: BOOL;								(* Start motion with constant velocity *)
	bMoveAbsolute			: BOOL;								(* Move to absolute position *)
	bMoveAdditive			: BOOL;								(* Move by distance *)
	bMoveRelative			: BOOL;								(* Move by distance *)
	bJog					: BOOL;								(* Start manual jog movement *)
	bStop					: BOOL;								(* High priority stop command *)
	bHalt					: BOOL;								(* Halt current motion, next motion command will abort this command *)
	bReset					: BOOL;								(* Reset axis and return to READY state *)
	
	(* General parameters *)
	bModulo					: BOOL;								(* Axis is periodic *)								
	lrOverride				: LREAL;							(* Axis velocity override in percents [%] *)
	lrVelocity 				: LREAL;							(* Axis velocirt in measurement units per second *)
	lrAcceleration			: LREAL;							(* Axis acceleration in measurement units per sercond^2 *)
	lrDeceleration 			: LREAL;							(* Axis deceleration in measurement units per sercond^2 *)
	lrJerk					: LREAL;							(* Axis jerk in measurement unit per sercond^3 *)
	lrAbsolutePosition		: LREAL;							(* Target position for MC_MoveAbsolute function *)
	lrRelativeDistance		: LREAL;							(* Relative distance to move for MC_MoveRelative/Additive fuctions *)
	lrHomePosition			: LREAL;							(* This parameters is used to set axis position while performing homing procedure *)
	
	(* Jog function parameters *)	
	lrJogPosition			: LREAL;							(* Relative position to move for jog feature *)
	lrJogVelocity			: LREAL;							(* Jog movement velocity *)
	lrJogAcceleration		: LREAL;							(* Jog movement acceleration *)
	lrJogDeceleration		: LREAL;							(* Jog movement deceleration *)
	lrJogJerk				: LREAL;							(* Jog movement jerk *)
	eJogMode				: E_JogMode;						(* Jog momement mode *)
	eJogDirection			: E_AxisJogDirection;				(* Direction of jog movement *)
	
	(* Stop function parameters *)
	lrStopDeceleration		: LREAL;							(* Stop deceleration *)
	lrStopJerk 				: LREAL;							(* Stop jerk *)
	
	(* Other parameters *)
	stOptions				: ST_MoveOptions;					(* Additional movement options *)
	eDirection				: Tc2_MC2.MC_Direction;				(* Axis movement direction for MC_MoveVelocity *)
	mcBufferMode 			: MC_BufferMode := MC_Aborting;		(* Axis buffering mode *)
	
	(* Axis status flags *)
	bActive					: BOOL;
	bBusy					: BOOL;								(* Function block currently executes one of the requests *)
	bError					: BOOL;								(* Error status flag *)
	iErrorID				: UDINT;							(* Error ID *)
	iAxisErrorID			: UDINT;							(* Axis error ID*)
	lrActualPosition		: LREAL;							(* Actual axis position in selected units *)
	rActualVelocity			: REAL;								(* Actual axis velocity in selected units *)
	bPowerOn 				: BOOL;								(* Power On status bit *)
	bIsHomed				: BOOL;								(* Axis has been homed even once *)
	bInVelocity				: BOOL;								(* Axis is moving in target velocity *)
	bInPostion				: BOOL;								(* Axis reached target position *)
	bMoveActive				: BOOL;								(* Axis is moving to target position *)
	bJogDone				: BOOL;								(* Axis manual movement by jog done *)
	bStopped				: BOOL;								(* Axis movement has been stopped *)
	bHalted					: BOOL;								(* Axis movement has been halted *)
	eStatePlcOpen			: E_AxisStatePlcOpen;				(* Current PLCOpen state of axis *)
	
	fbAxis					: FB_AxisJennyScienceEthercat;		(* Jenny Science axis instance *)
	
	bStartReversingSequence	: BOOL;								(* Starts sample reversing movement*)
	iReversingSequenceState : USINT;
	lrTargetPosition1		: LREAL := 5.0;
	lrTargetPosition2		: LREAL := 300.0;
	lrTargetVelocity		: LREAL := 200.0;
END_VAR

IF bFirstCycle THEN
	bFirstCycle := FALSE;
	
	fbAxis.MR_FirstCycle('Jenny Science Axis 1','mm', bModulo);
	
	lrOverride 			:= 100.0;
	lrVelocity 			:= 100.0;
	lrAcceleration		:= 1500.0;
	lrDeceleration		:= 1500.0;
	lrJerk				:= 1500.0;
	lrAbsolutePosition	:= 0.0;
	lrRelativeDistance	:= 0.0;
	lrHomePosition		:= 0.0;
	
	lrJogPosition		:= 0.0;
	lrJogVelocity 		:= 25.0;
	lrJogAcceleration	:= 250.0;
	lrJogDeceleration	:= 250.0;
	lrJogJerk			:= 250.0;
	
	lrStopDeceleration	:= 250.0;
	lrStopJerk			:= 250.0;
	
END_IF

bActive 			:= fbAxis.Active;
bBusy 				:= fbAxis.Busy;
bError 				:= fbAxis.Error;
iErrorID 			:= fbAxis.ErrorID;
iAxisErrorID 		:= fbAxis.ErrorID;
lrActualPosition 	:= fbAxis.ActualPosition;
rActualVelocity		:= fbAxis.ActualVelocity;
bPowerOn 			:= fbAxis.PowerOn;
bIsHomed 			:= fbAxis.IsHomed;
bInVelocity			:= fbAxis.InVelocity;
bInPostion 			:= fbAxis.InPosition;
bMoveActive 		:= fbAxis.MoveActive;
bJogDone 			:= fbAxis.JogDone;
bStopped 			:= fbAxis.Stopped;
bHalted 			:= fbAxis.Halted;
eStatePlcOpen 		:= fbAxis.StatePlcOpen;

IF bReset THEN
	IF fbAxis.MR_Reset() THEN
		bReset := FALSE;
	END_IF
END_IF

(* Stop commands *)
IF bStop THEN
	bJog := FALSE;
	bMoveAbsolute := FALSE;
	bMoveAdditive := FALSE;
	bMoveRelative := FALSE;
	bMoveVelocity := FALSE;
	iReversingSequenceState := 0;
	
	fbAxis.MR_Stop();
	IF fbAxis.Stopped THEN
		bStop := FALSE;
	END_IF
	
ELSIF bHalt THEN
	bJog := FALSE;
	bMoveAbsolute := FALSE;
	bMoveAdditive := FALSE;
	bMoveRelative := FALSE;
	bMoveVelocity := FALSE;
	iReversingSequenceState := 0;
	
	fbAxis.MR_Halt();
	IF fbAxis.Halted THEN
		bHalt := FALSE;
	END_IF
	
END_IF

(* Other commands *)
IF bInit THEN	
	fbAxis.MR_Init();	
	IF fbAxis.PowerOn THEN
		bInit := FALSE;
	END_IF
	
ELSIF bDeinit THEN
	fbAxis.MR_Abort();
	IF NOT fbAxis.PowerOn THEN
		bDeinit := FALSE;
	END_IF
	
ELSIF bHome THEN
	fbAxis.MR_Home(lrHomePosition);
	IF fbAxis.IsHomed THEN
		bHome := FALSE;
	END_IF
	
ELSIF bMoveVelocity THEN
	fbAxis.MR_MoveVelocity();
	IF fbAxis.InVelocity THEN
		bMoveVelocity := FALSE;
	END_IF
	
ELSIF bMoveAbsolute THEN
	fbAxis.MR_MoveAbsolute(lrAbsolutePosition);
	IF fbAxis.InPosition THEN
		bMoveAbsolute := FALSE;
	END_IF

ELSIF bMoveAdditive THEN
	fbAxis.MR_MoveAdditive(lrRelativeDistance);
	IF fbAxis.InPosition THEN
		bMoveAdditive := FALSE;
	END_IF
	
ELSIF bMoveRelative THEN
	fbAxis.MR_MoveRelative(lrRelativeDistance);
	IF fbAxis.InPosition THEN
		bMoveRelative := FALSE;
	END_IF
	
ELSIF bJog THEN
	(*fbAxis.MR_Jog(lrJogPosition,eJogDirection);
	IF fbAxis.JogDone THEN
		bJog := FALSE;	
	END_IF
	*)
	
	fbAxis.MR_Jog(bJog);
	bJog:= FALSE;
	
END_IF

CASE iReversingSequenceState OF
	(* Starts seqence *)
	0:
		IF bStartReversingSequence THEN
			bStartReversingSequence := FALSE;
			iReversingSequenceState := 10;
		END_IF	
		
	(* Move to first postion *)
	10:
		lrVelocity := lrTargetVelocity;
		fbAxis.MR_MoveAbsolute(lrTargetPosition1);
		IF fbAxis.InPosition THEN
			iReversingSequenceState := 20;
		END_IF
		
	(* Move to second position *)
	20:
		lrVelocity := lrTargetVelocity;
		fbAxis.MR_MoveAbsolute(lrTargetPosition2);
		IF fbAxis.InPosition THEN
			iReversingSequenceState := 10;
		END_IF
		
END_CASE

fbAxis.Override 		:= lrOverride;
fbAxis.Velocity 		:= lrVelocity;
fbAxis.Acceleration		:= lrAcceleration;
fbAxis.Deceleration 	:= lrDeceleration;
fbAxis.Jerk 			:= lrJerk;
fbAxis.JogVelocity 		:= lrJogVelocity;
fbAxis.JogAcceleration 	:= lrJogAcceleration;
fbAxis.JogDeceleration 	:= lrJogDeceleration;
fbAxis.JogJerk 			:= lrJogJerk;
fbAxis.StopDeceleration := lrStopDeceleration;
fbAxis.StopJerk 		:= lrStopJerk;

fbAxis();

END_PROGRAM

// ---- POUs/Universal Blocks/Axis/PRG_FB_AxisServo_Test.TcPOU
PROGRAM PRG_FB_AxisServo_Test
VAR
	bFirstCycle 	: BOOL := TRUE;
	
	bInit					: BOOL;								(* Power on axis and prepare to work *)
	bAbort					: BOOL;								(* Power off axis and reset status flags *)
	bHome					: BOOL;								(* Home to reference point *)
	bMoveVelocity			: BOOL;								(* Start motion with constant velocity *)
	bMoveAbsolute			: BOOL;								(* Move to absolute position *)
	bMoveAdditive			: BOOL;								(* Move by distance *)
	bMoveRelative			: BOOL;								(* Move by distance *)
	bJog					: BOOL;								(* Start manual jog movement *)
	bStop					: BOOL;								(* High priority stop command *)
	bHalt					: BOOL;								(* Halt current motion, next motion command will abort this command *)
	bReset					: BOOL;								(* Reset axis and return to READY state *)
	
	(* General parameters *)
	bModulo					: BOOL := FALSE;					(* Axis is periodic *)
	lrOverride				: LREAL;							(* Axis velocity override in percents [%] *)
	lrVelocity 				: LREAL;							(* Axis velocirt in measurement units per second *)
	lrAcceleration			: LREAL;							(* Axis acceleration in measurement units per sercond^2 *)
	lrDeceleration 			: LREAL;							(* Axis deceleration in measurement units per sercond^2 *)
	lrJerk					: LREAL;							(* Axis jerk in measurement unit per sercond^3 *)
	lrAbsolutePosition		: LREAL;							(* Target position for MC_MoveAbsolute function *)
	lrRelativeDistance		: LREAL;							(* Relative distance to move for MC_MoveRelative/Additive fuctions *)
	lrHomePosition			: LREAL;							(* This parameters is used to set axis position while performing homing procedure *)
	
	(* Jog function parameters *)	
	lrJogPosition			: LREAL;							(* Relative position to move for jog feature *)
	lrJogVelocity			: LREAL;							(* Jog movement velocity *)
	lrJogAcceleration		: LREAL;							(* Jog movement acceleration *)
	lrJogDeceleration		: LREAL;							(* Jog movement deceleration *)
	lrJogJerk				: LREAL;							(* Jog movement jerk *)
	eJogMode				: E_JogMode;						(* Jog movement mode *)
	eJogDirection			: E_AxisJogDirection;				(* Direction of jog movement *)
	
	(* Stop function parameters *)
	lrStopDeceleration		: LREAL;							(* Stop deceleration *)
	lrStopJerk 				: LREAL;							(* Stop jerk *)
	
	(* Other parameters *)
	stOptions				: ST_MoveOptions;					(* Additional movement options *)
	eDirection				: Tc2_MC2.MC_Direction;				(* Axis movement direction for MC_MoveVelocity *)
	eBufferMode 			: MC_BufferMode := MC_Aborting;		(* Axis buffering mode *)
	
	(* Axis status flags *)
	bActive					: BOOL;
	bBusy					: BOOL;								(* Function block currently executes one of the requests *)
	bError					: BOOL;								(* Error status flag *)
	iErrorID				: UDINT;							(* Error ID *)
	iAxisErrorID			: UDINT;							(* Axis error ID*)
	lrActualPosition		: LREAL;							(* Actual axis position in selected units *)
	rActualVelocity			: REAL;								(* Actual axis velocity in selected units *)
	bPowerOn 				: BOOL;								(* Power On status bit *)
	bIsHomed				: BOOL;								(* Axis has been homed even once *)
	bInVelocity				: BOOL;								(* Axis is moving in target velocity *)
	bInPostion				: BOOL;								(* Axis reached target position *)
	bMoveActive				: BOOL;								(* Axis is moving to target position *)
	bJogDone				: BOOL;								(* Axis manual movement by jog done *)
	bStopped				: BOOL;								(* Axis movement has been stopped *)
	bHalted					: BOOL;								(* Axis movement has been halted *)
	eStatePlcOpen			: E_AxisStatePlcOpen;				(* Current PLCOpen state of axis *)
	
	fbAxis					: FB_AxisServo;
	
	iAxisStateMachine		: INT;
END_VAR

IF bFirstCycle THEN
	bFirstCycle := FALSE;
	fbAxis.MR_FirstCycle('Standard Beckhoff Axis 1','deg',bModulo);
	
	lrOverride 			:= 100.0;
	lrVelocity 			:= 100.0;
	lrAcceleration		:= 1500.0;
	lrDeceleration		:= 1500.0;
	lrJerk				:= 1500.0;
	lrAbsolutePosition	:= 0.0;
	lrRelativeDistance	:= 0.0;
	lrHomePosition		:= 0.0;
	
	lrJogPosition		:= 0.0;
	lrJogVelocity 		:= 25.0;
	lrJogAcceleration	:= 250.0;
	lrJogDeceleration	:= 250.0;
	lrJogJerk			:= 250.0;
	
	lrStopDeceleration	:= 250.0;
	lrStopJerk			:= 250.0;	
END_IF

bActive 			:= fbAxis.Active;
bBusy				:= fbAxis.Busy;
bError 				:= fbAxis.Error;
iErrorID 			:= fbAxis.ErrorID;
iAxisErrorID 		:= fbAxis.ErrorID;
lrActualPosition 	:= fbAxis.ActualPosition;
rActualVelocity		:= fbAxis.ActualVelocity;
bPowerOn 			:= fbAxis.PowerOn;
bIsHomed 			:= fbAxis.IsHomed;
bInVelocity			:= fbAxis.InVelocity;
bInPostion 			:= fbAxis.InPosition;
bMoveActive 		:= fbAxis.MoveActive;
bJogDone 			:= fbAxis.JogDone;
bStopped 			:= fbAxis.Stopped;
bHalted 			:= fbAxis.Halted;
eStatePlcOpen		:= fbAxis.StatePlcOpen;

IF bStop THEN
	bStop := FALSE;
	iAxisStateMachine := 20;
	
ELSIF bHalt THEN
	bHalt := FALSE;
	iAxisStateMachine := 30;
	
ELSIF bReset THEN
	bReset := FALSE;
	iAxisStateMachine := 40;
	
ELSIF bAbort THEN
	bAbort := FALSE;
	iAxisStateMachine := 110;
	
END_IF

CASE iAxisStateMachine OF
	(* Starts seqence *)
	0:
		IF bInit THEN
			bInit := FALSE;
			iAxisStateMachine := 10;

		ELSIF bHome THEN
			bHome := FALSE;
			iAxisStateMachine := 50;
			
		ELSIF bMoveVelocity THEN
			bMoveVelocity := FALSE;
			iAxisStateMachine := 60;
		
		ELSIF bMoveAbsolute THEN
			bMoveAbsolute := FALSE;
			iAxisStateMachine := 70;
		
		ELSIF bMoveAdditive THEN
			bMoveAdditive := FALSE;
			iAxisStateMachine := 80;
			
		ELSIF bMoveRelative THEN
			bMoveRelative := FALSE;
			iAxisStateMachine := 90;
			
		ELSIF bJog THEN
			iAxisStateMachine := 100;
		
		END_IF
		
	(* Initialization *)
	10:
		fbAxis.MR_Init();	
		IF fbAxis.PowerOn THEN
			iAxisStateMachine := 0;
		END_IF
		
	(* Stopping *)
	20:
		bJog := FALSE;
		bMoveAbsolute := FALSE;
		bMoveAdditive := FALSE;
		bMoveRelative := FALSE;
		bMoveVelocity := FALSE;
		
		IF fbAxis.MR_Stop() THEN
			iAxisStateMachine := 0;
		END_IF
		
	(* Halting *)
	30:
		bJog := FALSE;
		bMoveAbsolute := FALSE;
		bMoveAdditive := FALSE;
		bMoveRelative := FALSE;
		bMoveVelocity := FALSE;
		
		fbAxis.MR_Halt();
		IF fbAxis.Halted THEN
			iAxisStateMachine := 0;
		END_IF
		
	(* Resetting *)
	40:
		fbAxis.MR_Reset(); 
		IF NOT fbAxis.Error THEN
			iAxisStateMachine := 0;
		END_IF
	
	(* Homing *)
	50: 
		fbAxis.MR_Home(lrHomePosition);
		IF fbAxis.IsHomed THEN
			iAxisStateMachine := 0;
		END_IF
	
	(* Move velocity *)	
	60: 
		fbAxis.MR_MoveVelocity();
		IF fbAxis.InVelocity THEN
			iAxisStateMachine := 0;
		END_IF	
		
	(* Move absolute *)	
	70: 
		fbAxis.MR_MoveAbsolute(lrAbsolutePosition);
		IF fbAxis.InPosition THEN
			iAxisStateMachine := 0;
		END_IF
		
	(* Move additive *)	
	80: 
		fbAxis.MR_MoveAdditive(lrRelativeDistance);
		IF fbAxis.InPosition THEN
			iAxisStateMachine := 0;
		END_IF
		
	(* Move relative *)	
	90: 
		fbAxis.MR_MoveRelative(lrRelativeDistance);
		IF fbAxis.InPosition THEN
			iAxisStateMachine := 0;
		END_IF
		
	(* Jog movement *)	
	100: 
		fbAxis.MR_Jog(bJog);
		IF fbAxis.JogDone THEN
			bJog := FALSE;
			iAxisStateMachine := 0;
		END_IF
		
	(* Deinitialization *)	
	110: 
		fbAxis.MR_Abort();
		IF NOT fbAxis.PowerOn THEN
			iAxisStateMachine := 0;
		END_IF		
END_CASE

fbAxis.Override			:= lrOverride;
fbAxis.Velocity 		:= lrVelocity;
fbAxis.Acceleration 	:= lrAcceleration;
fbAxis.Deceleration 	:= lrDeceleration;
fbAxis.Jerk 			:= lrJerk;
fbAxis.JogMode			:= eJogMode;
fbAxis.JogDirection		:= eJogDirection;
fbAxis.JogVelocity 		:= lrJogVelocity;
fbAxis.JogAcceleration 	:= lrJogAcceleration;
fbAxis.JogDeceleration 	:= lrJogDeceleration;
fbAxis.JogJerk 			:= lrJogJerk;
fbAxis.StopDeceleration := lrStopDeceleration;
fbAxis.StopJerk 		:= lrStopJerk;

fbAxis();

END_PROGRAM

// ---- POUs/Universal Blocks/Communication/Backhoff ADS/PRG_FB_AdsExchanger_Test.TcPOU
PROGRAM PRG_FB_AdsExchanger_Test
VAR
	bFirstCycle 	: BOOL := TRUE;
	bInit 			: BOOL;
	bDeinit 		: BOOL;
	bRead 			: BOOL;
	bWritte 		: BOOL;
	bReset 			: BOOL;
	
	sAmsNetID		: STRING	:= '5.68.97.76.1.1';
	iAmsPort 		: UINT 		:= 851;
	iIndexGroup 	: UDINT 	:= 16#4020;
	iIndexOffset	: UDINT 	:= 0;
	
	bActive			: BOOL;
	bBusy			: BOOL;
	bError			: BOOL;
	iErrorID		: UDINT;
	iAdsErrorID 	: UDINT;
	State 			: E_AdsExchangerState;
	
	sReadMessage 	: STRING;
	sWritteMessage 	: STRING;
	
	fbAdsExchanger	: FB_AdsExchanger;
END_VAR

IF bFirstCycle THEN
	bFirstCycle := FALSE;
	fbAdsExchanger.MR_FirstCycle('My test ADS exchanger', sAmsNetID, iAmsPort);
END_IF

bActive := fbAdsExchanger.Active;
bBusy := fbAdsExchanger.Busy;
bError := fbAdsExchanger.Error;
iErrorID := fbAdsExchanger.ErrorID;
State := fbAdsExchanger.State;

IF bInit THEN
	IF fbAdsExchanger.MR_Init() THEN
		bInit := FALSE;
	END_IF
	
ELSIF bDeinit THEN
	IF fbAdsExchanger.MR_Abort() THEN
		bDeinit := FALSE;
	END_IF
	
ELSIF bRead THEN
	IF fbAdsExchanger.MR_Read(ADR(sReadMessage)) THEN
		bRead := FALSE;
	END_IF
	
ELSIF bWritte THEN
	IF fbAdsExchanger.MR_Writte(ADR(sWritteMessage)) THEN
		bWritte := FALSE;
	END_IF
	
ELSIF bReset THEN
	IF fbAdsExchanger.MR_Reset() THEN
		bReset := FALSE;
	END_IF
	
END_IF

fbAdsExchanger.AmsNetID		:= sAmsNetID;
fbAdsExchanger.AmsPort 		:= iAmsPort;
fbAdsExchanger.IndexGroup 	:= iIndexGroup;
fbAdsExchanger.IndexOffset 	:= iIndexOffset;

fbAdsExchanger();

END_PROGRAM

// ---- POUs/Universal Blocks/Communication/TcpIp/PRG_FB_TcpClient_Test.TcPOU
PROGRAM PRG_FB_TcpClient_Test
VAR
	bFirstCycle 		: BOOL := TRUE;
	fbTcpClient 		: FB_TcpClient;
	fbFileLogger		: FB_FileLogger; 
	
	iState 				: USINT;
	
	bInit 				: BOOL;
	bAbort 				: BOOL;
	bNewPar				: BOOL;
	bSend 				: BOOL;
	bRecive 			: BOOL;
	bReciveAndSend		: BOOL;
	
	sSendMessage 		: STRING;
	sSendMessage1		: STRING;
	sReciveMessage 		: STRING;

	bError				: BOOL;
	iErrorID			: UDINT;
	eClientState		: E_TcpIpDeviceState;
	
	sHost				: T_IPv4Addr;
	iPort				: UINT;
	
	stSendData 			: ST_TcpBufferData;
	stReciveData 		: ST_TcpBufferData;
	
	arrBufferMessage	: ARRAY[0..10] OF STRING;
	iMessageIndex	 	: INT;
	bArrBufferClear 	: BOOL;
	
	sDirectoryForSimulation : STRING := 'C:\TwinCAT\Tests\';
	
	tAddLogg : TON;
	
END_VAR

(* Setting initial parameters *)
IF bFirstCycle THEN
	bFirstCycle := FALSE;
	fbTcpClient.MR_FirstCycle(	sName		:= 'TCP/IP test client',
								sHost 		:= '192.168.0.100',
								sAmsNetID	:= '',
								iPort		:= 12000,
								tTimeout	:= T#5S);
								
	fbFileLogger.MR_FirstCycle( sName		:= 'File Logger',
								sFileDir 	:= sDirectoryForSimulation,
								sFileName 	:= 'LoggerVisionTest',
								sAmsNetId 	:= '',
								bAddTimeStamp := TRUE,
								bAddHeader := TRUE);	
	iState := 0;
END_IF

bError := fbTcpClient.Error;
iErrorID := fbTcpClient.ErrorID;
eClientState := fbTcpClient.State;


(* Closing the client connection *)
IF bAbort THEN
	bAbort := FALSE;
	iState := 20;
END_IF

(* Setting new parameters before initialization*)
IF bNewPar THEN
	bNewPar := FALSE;
	fbTcpClient.Host := sHost;
	fbTcpClient.Port := iPort;
END_IF

CASE iState OF
	(* Waiting for commands *)
	0:
		IF bInit THEN
			bInit := FALSE;
		//	fbFileLogger.MR_Init();
		//	IF fbFileLogger.Active THEN
				iState := 10;
		//	END_IF

		ELSIF bSend THEN
			bSend := FALSE;
			iState := 30;
			
		ELSIF bRecive THEN
			IF NOT bArrBufferClear THEN
				iState := 60;
			ELSE
				bArrBufferClear := 0;
				bRecive := FALSE;
				iState := 40;
			END_IF
		
		ELSIF bReciveAndSend THEN
			bReciveAndSend := FALSE;
			iState := 45;
			
		END_IF
		
	(* Client connection initialization *)
	10:
		fbTcpClient.MR_Init();
		IF fbTcpClient.Active THEN
			iState := 0;
		END_IF
		
	(* Client connection deinitialization *)
	20:
		fbTcpClient.MR_Abort();
		IF NOT fbTcpClient.Active THEN
			iState := 0;	
		END_IF
	
	(* Sending messages *)
	30:
		MEMCPY(ADR(sSendMessage1),ADR(sSendMessage),SIZEOF(sSendMessage));
		sSendMessage := CONCAT(sSendMessage, ':1$N');
		FUN_StringToTcpBufferData(ADR(sSendMessage),ADR(stSendData));
		
		IF fbTcpClient.MR_AppendToSendBuffer(stSendData) THEN
			sSendMessage := CONCAT(sSendMessage1, ':2$N');
			FUN_StringToTcpBufferData(ADR(sSendMessage1),ADR(stSendData));
			
			IF fbTcpClient.MR_AppendToSendBuffer(stSendData) THEN
				iState := 50;
			END_IF
		END_IF
		
	(* Receiving messages to array buffer *)
	40:
		stReciveData := fbTcpClient.NextRecivedMessage;
		IF stReciveData.iLength > 0 THEN
			FUN_TcpBufferDataToString(ADR(sReciveMessage),ADR(stReciveData));
			arrBufferMessage[iMessageIndex] := sReciveMessage;
			iMessageIndex := iMessageIndex + 1;
		ELSIF stReciveData.iLength = 0 THEN
			iMessageIndex := 0;
			iState := 0;

		END_IF
		
	(* Sending last received message *)
	45:
		stReciveData := fbTcpClient.LastRecivedMessage;
		IF stReciveData.iLength > 0 THEN
			FUN_TcpBufferDataToString(ADR(sReciveMessage),ADR(stReciveData));
			sSendMessage := CONCAT('Response to: ',sReciveMessage);
			sSendMessage := CONCAT(sSendMessage, '$N');
			FUN_StringToTcpBufferData(ADR(sSendMessage),ADR(stSendData));
			iState := 30;
			
		END_IF	
		
	(* Clearing buffers *)
	50:
		fbTcpClient.MR_ClearAllBuffers();
		iState := 0;
		
	(* Clearing incoming messages array buffer *)
	60:
		bArrBufferClear := TRUE;
		MEMSET(ADR(arrBufferMessage), 0, SIZEOF(arrBufferMessage));
		iState := 0;
		
END_CASE

fbTcpClient();
fbFileLogger();
tAddLogg();

END_PROGRAM

// ---- POUs/Universal Blocks/Communication/TcpIp/PRG_FB_TcpServer_Test.TcPOU
PROGRAM PRG_FB_TcpServer_Test
VAR
	iAdr			: PVOID;
	bFristCycle 	: BOOL := TRUE;			(*  *)
	fbTcpServer		: FB_TcpServer;			(*  *)
	fbFileLogger	: FB_FileLogger; 
	
	iServerState 	: USINT;				(*  *)
	
	bInit 			: BOOL;					(*  *)
	bAbort 			: BOOL;					(*  *)
	bDisconnect		: BOOL;					(*  *)
	
	sSendMessage 	: STRING;				(*  *)
	sReciveMessage	: STRING;				(*  *)
	
	bError			: BOOL;					(*  *)
	iErrorID		: UDINT;				(*  *)
	eState			: E_TcpIpDeviceState; 	(*  *)
	eServerState	: E_TcpIpServerStateRunning;	(*  *)
	iState			: USINT;
	
	stSendData		: ST_TcpBufferData;		(*  *)
	stReciveData 	: ST_TcpBufferData;		(*  *)
	
	sDirectoryForSimulation : STRING := 'C:\TwinCAT\Tests\';
	
	tAddLogg : TON;
	
END_VAR

(* Setting initial parameters *)
IF bFristCycle THEN
	bFristCycle := FALSE;
	fbTcpServer.MR_FirstCycle(	sName		:= 'TCP/IP test server',
								sHost		:= '',
								sAmsNetID	:= '',
								iPort		:= 12000,
								tTimeout	:= T#10S);
								
	fbFileLogger.MR_FirstCycle( sName		:= 'File Logger',
								sFileDir 	:= sDirectoryForSimulation,
								sFileName 	:= 'LoggerVisionTest',
								sAmsNetId 	:= '',
								bAddTimeStamp := TRUE,
								bAddHeader := TRUE);							
	
END_IF

bError 			:= fbTcpServer.Error;
iErrorID 		:= fbTcpServer.ErrorID;
eState 			:= fbTcpServer.State;
eServerState 	:= fbTcpServer.ServerState;

(* Closing the server *)
IF bAbort THEN
	bAbort := FALSE;
	iState := 40;
END_IF

CASE iState OF
	(* Server not ready waiting for init command *)
	0:
		IF bInit THEN
			bInit := FALSE;
			fbFileLogger.MR_Init();
			IF fbFileLogger.Active THEN
				iState := 10;
			END_IF
		END_IF
	
	(* Server initialization*)	
	10:
		fbTcpServer.MR_Init();
		IF fbTcpServer.Active THEN
			bInit := FALSE;
			iState := 20;
		END_IF
		
	(* Server is running - waiting for client and data exchange *)	
	20:
		IF fbTcpServer.ServerState = TCPIP_SERVER_RUNNING_DATA_EXCHANGE THEN
			stReciveData := fbTcpServer.LastRecivedMessage;	
		
			IF bDisconnect THEN
				bDisconnect := FALSE;
				iState := 30;
			
			ELSIF stReciveData.iLength > 0 THEN
				FUN_TcpBufferDataToString(ADR(sReciveMessage),ADR(stReciveData));
				iState := 22;
			END_IF
		END_IF
		
	22:
		FUN_StringToTcpBufferData(ADR(sReciveMessage),ADR(stSendData));
		fbTcpServer.MR_AppendToSendBuffer(stReciveData);
		iState := 25;	
	25:
		fbTcpServer.MR_ClearAllBuffers();
		iState := 20;
	
	(* Disconnecting from current connection*)
	30:
		fbTcpServer.MR_Disconnect();
		
		IF fbTcpServer.ServerState = TCPIP_SERVER_RUNNING_CLOSE_CONNECTION_DONE THEN
			iState := 20;
		END_IF
	(* Server deinitialization *)
	40:
		fbTcpServer.MR_Abort();
		
		IF NOT fbTcpServer.Active THEN
			iState := 0;
		END_IF
	
END_CASE

fbTcpServer();
fbTcpServer();
fbFileLogger();
fbFileLogger();
tAddLogg();

END_PROGRAM

// ---- POUs/Universal Blocks/Communication/TcpIp/PRG_FUN_TcpDataConversion_Test.TcPOU
PROGRAM PRG_FUN_TcpDataConversion_Test
VAR
	bConvert 			: BOOL;
	bRevert				: BOOL;
	bConversionResult 	: BOOL;
	bReversionResult	: BOOL;
	sSendMessage		: STRING;
	sRecivedMessage 	: STRING;
	stSendData 			: ST_TcpBufferData;
END_VAR

IF bConvert THEN
	bConversionResult := FUN_StringToTcpBufferData(ADR(sSendMessage),ADR(stSendData));
	IF bConversionResult THEN
		bConvert := FALSE;
	END_IF
	
ELSIF bRevert THEN
	bReversionResult := FUN_TcpBufferDataToString(ADR(sRecivedMessage),ADR(stSendData));
	IF bReversionResult THEN
		bRevert := FALSE;
	END_IF
END_IF

END_PROGRAM

// ---- POUs/Universal Blocks/Cylinder/PRG_FB_SingleCoilCylinder_Test.TcPOU
PROGRAM PRG_FB_SingleCoilCylinder_Test
VAR
	bFirstCycle : BOOL := TRUE;
	
	(* Commands *)
	bInit			: BOOL;					(* Cylinder init command *)
	bAbort			: BOOL;					(* Cylinder deinit command *)
	bGoHome			: BOOL;					(* Go to home position command *)
	bGoActive		: BOOL;					(* Go to active position command *)
	bRelease		: BOOL;					(* Cylinder release command *)
	bReset			: BOOL;					(* Cylinder reset command *)
	
	(* Parameters *)
	tDelay			: TIME := T#100MS;		(*  *)
	tActiveTimeout	: TIME := T#20S;		(*  *)
	tHomeTimeout	: TIME := T#20S;		(*  *)
	bSimulation 	: BOOL := FALSE;		(* Simulation enable bit *)
	
	(* Status *)
	bActive			: REFERENCE TO BOOL;				(*  *)
	bBusy			: REFERENCE TO BOOL;				(*  *)
	bError			: REFERENCE TO BOOL;				(*  *)
	eErrorID		: REFERENCE TO E_CylinderError;		(*  *)
	tMoveActiveTime	: REFERENCE TO TIME;				(*  *)
	tMoveHomeTime	: REFERENCE TO TIME;				(*  *)
	bSensorHome		: REFERENCE TO BOOL;				(* Sensor home status bit *)
	bSensorActive 	: REFERENCE TO BOOL;				(* Sensor active status bit *)
	bPostionHold	: REFERENCE TO BOOL;				(* Set true if position of cylinder is held by pressure *)
	eState			: REFERENCE TO E_CylinderState;		(*  *)
	
	iState			: USINT;
	
	(* FB's*)
	fbTestCylinder : FB_SingleCoilCylinder;				(* Single coil cylinder object *)
	
END_VAR

IF bFirstCycle THEN
	bFirstCycle := FALSE;
	fbTestCylinder.MR_FirstCycle( 	sName := 'Single_Coil_Cylinder',
									tGoHomeTimeout := T#10S,
									tGoActiveTimeout := T#10S,
									tDelay := tDelay);
									
									
	bActive			REF= fbTestCylinder.Active;
	bBusy			REF= fbTestCylinder.Busy;
	bError 			REF= fbTestCylinder.Error;
	eErrorID 		REF= fbTestCylinder.ErrorID;
	eState			REF= fbTestCylinder.State;
	tMoveActiveTime REF= fbTestCylinder.MoveActiveTime;
	tMoveHomeTime 	REF= fbTestCylinder.MoveHomeTime;
	bSensorHome 	REF= fbTestCylinder.PositionHome;
	bSensorActive 	REF= fbTestCylinder.PositionActive;
	bPostionHold	REF= fbTestCylinder.PositionHold;
END_IF

(* Simple controler *)
IF bReset THEN
	bReset := FALSE;
	iState := 60;
	
ELSIF bAbort THEN
	bAbort := FALSE;
	iState := 20;
	
END_IF

CASE iState OF
	0:
		IF bInit THEN
			bInit := FALSE;
			iState := 10;
			
		ELSIF bGoHome THEN
			bGoHome := FALSE;
			iState := 30;
			
		ELSIF bGoActive THEN
			bGoActive := FALSE;
			iState := 40;
			
		ELSIF bRelease THEN
			bRelease := FALSE;
			iState := 50;
			
		END_IF
	10:
		fbTestCylinder.MR_Init();
		
		IF fbTestCylinder.Active THEN
			iState := 0;
		END_IF
	20:
		fbTestCylinder.MR_Abort();
		
		IF NOT fbTestCylinder.Active THEN
			iState := 0;
		END_IF
	30:
		fbTestCylinder.MR_GoHome();
		
		IF fbTestCylinder.PositionHome AND NOT fbTestCylinder.Busy THEN
			iState := 0;
		END_IF
	40:
		fbTestCylinder.MR_GoActive();
		
		IF fbTestCylinder.PositionActive AND NOT fbTestCylinder.Busy THEN
			iState := 0;
		END_IF
	50:
		fbTestCylinder.MR_Release();
		
		IF NOT fbTestCylinder.PositionHold AND NOT fbTestCylinder.Busy THEN
			iState := 0;
		END_IF
	60:
		fbTestCylinder.MR_Reset();
		
		IF NOT fbTestCylinder.Error THEN
			iState := 0;
		END_IF
		
END_CASE

fbTestCylinder.Simulation := bSimulation;
fbTestCylinder.Delay := tDelay;
fbTestCylinder.ActiveTimeout := tActiveTimeout;
fbTestCylinder.HomeTimeout := tHomeTimeout;
fbTestCylinder();

END_PROGRAM

// ---- POUs/Universal Blocks/Cylinder/PRG_FB_DoubleCoilCylinder_Test.TcPOU
PROGRAM PRG_FB_DoubleCoilCylinder_Test
VAR
	bFirstCycle : BOOL := TRUE;
	(* Commands *)
	bInit			: BOOL;					(* Cylinder init command *)
	bAbort			: BOOL;					(* Cylinder deinit command *)
	bGoHome			: BOOL;					(* Go to home position command *)
	bGoActive		: BOOL;					(* Go to active position command *)
	bRelease		: BOOL;					(* Cylinder release command *)
	bReset			: BOOL;					(* Cylinder reset command *)
	
	(* Parameters *)
	tDelay			: TIME := T#100MS;		(*  *)
	tActiveTimeout	: TIME := T#20S;		(*  *)
	tHomeTimeout	: TIME := T#20S;		(*  *)
	bSimulation 	: BOOL := TRUE;			(* Simulation enable bit *)
	
	(* Status *)
	bActive			: REFERENCE TO BOOL;				(*  *)
	bBusy			: REFERENCE TO BOOL;				(*  *)
	bError			: REFERENCE TO BOOL;				(*  *)
	eErrorID		: REFERENCE TO E_CylinderError;		(*  *)
	tMoveActiveTime	: REFERENCE TO TIME;				(*  *)
	tMoveHomeTime	: REFERENCE TO TIME;				(*  *)
	bSensorHome		: REFERENCE TO BOOL;				(* Sensor home status bit *)
	bSensorActive 	: REFERENCE TO BOOL;				(* Sensor active status bit *)
	eState			: REFERENCE TO E_CylinderState;		(*  *)
	
	fbTestCylinder : FB_DoubleCoilCylinder;	(* Universal cylinder object *)	
	iState: USINT;
END_VAR

IF bFirstCycle THEN
	bFirstCycle := FALSE;
	fbTestCylinder.MR_FirstCycle( 	sName := 'Double_Coil_Cylinder',
									tGoHomeTimeout := T#10S,
									tGoActiveTimeout := T#10S,
									tDelay := tDelay);
									
	bActive			REF= fbTestCylinder.Active;
	bBusy			REF= fbTestCylinder.Busy;
	bError 			REF= fbTestCylinder.Error;
	eErrorID 		REF= fbTestCylinder.ErrorID;
	eState			REF= fbTestCylinder.State;
	tMoveActiveTime REF= fbTestCylinder.MoveActiveTime;
	tMoveHomeTime 	REF= fbTestCylinder.MoveHomeTime;
	bSensorHome 	REF= fbTestCylinder.PositionHome;
	bSensorActive 	REF= fbTestCylinder.PositionActive;
END_IF

(* Simple controler *)
IF bReset THEN
	bReset := FALSE;
	iState := 60;
	
ELSIF bAbort THEN
	bAbort := FALSE;
	iState := 20;
	
END_IF

CASE iState OF
	0:
		IF bInit THEN
			bInit := FALSE;
			iState := 10;
			
		ELSIF bGoHome THEN
			bGoHome := FALSE;
			iState := 30;
			
		ELSIF bGoActive THEN
			bGoActive := FALSE;
			iState := 40;
			
		ELSIF bRelease THEN
			bRelease := FALSE;
			iState := 50;
			
		END_IF
	10:
		fbTestCylinder.MR_Init();
		
		IF fbTestCylinder.Active THEN
			iState := 0;
		END_IF
	20:
		fbTestCylinder.MR_Abort();
		
		IF NOT fbTestCylinder.Active THEN
			iState := 0;
		END_IF
	30:
		fbTestCylinder.MR_GoHome();
		
		IF fbTestCylinder.PositionHome AND NOT fbTestCylinder.Busy THEN
			iState := 0;
		END_IF
	40:
		fbTestCylinder.MR_GoActive();
		
		IF fbTestCylinder.PositionActive AND NOT fbTestCylinder.Busy THEN
			iState := 0;
		END_IF
	50:
		fbTestCylinder.MR_Release();
		
		IF NOT fbTestCylinder.PositionHold AND NOT fbTestCylinder.Busy THEN
			iState := 0;
		END_IF
	60:
		fbTestCylinder.MR_Reset();
		
		IF NOT fbTestCylinder.Error THEN
			iState := 0;
		END_IF
		
END_CASE

fbTestCylinder.Simulation := bSimulation;
fbTestCylinder.Delay := tDelay;
fbTestCylinder.ActiveTimeout := tActiveTimeout;
fbTestCylinder.HomeTimeout := tHomeTimeout;
fbTestCylinder();

END_PROGRAM

// ---- POUs/Universal Blocks/Digital Devices/Beacon/PRG_FB_Beacon_Test.TcPOU
PROGRAM PRG_FB_Beacon_Test
VAR CONSTANT
	sBEACON_NAME	: STRING := 'Electrical_Cabinet_Beacon';
END_VAR
VAR	
	bFirstCycle		: BOOL;
	
	(* Parameters *)
	bAnyError 		: BOOL;					(* Error status bit *)
	bAnyWarrning 	: BOOL;					(* Warrning status bit *)
	bReady 			: BOOL;					(* Machine ready status bit *)
	bRunning 		: BOOL;					(* Machine running status bit *)
	tFlashingTime 	: TIME := T#500MS;		(* Flashing time of red lamp *)
	
	(* FB's *)
	fbBeacon  		: FB_Beacon;			(* Beacon object *)
END_VAR

IF bFirstCycle THEN
	bFirstCycle := FALSE;
	fbBeacon.MR_FirstCycle( sName := sBEACON_NAME);
END_IF

fbBeacon.AnyError		:= bAnyError;
fbBeacon.AnyWarrning 	:= bAnyWarrning;
fbBeacon.Ready 			:= bReady;
fbBeacon.Running 		:= bRunning;

fbBeacon.RedLampFlashingTime := tFlashingTime;
fbBeacon();

END_PROGRAM

// ---- POUs/Universal Blocks/Digital Devices/Digital Input/PRG_FB_DigitalInput_Test.TcPOU
PROGRAM PRG_FB_DigitalInput_Test
VAR	
	bFirstCycle : BOOL := TRUE;
	
	bValue					: BOOL;				(* Current value of input from object *)
	bEnableForce			: BOOL;				(* Enables forcing in digital input object *)
	bFallingTrigger			: BOOL;				(* Falling trigger detected bit *)
	bRisingTrigger			: BOOL;				(* Rising trigger detected bit *)
	bSetForceValue			: BOOL;				(* Triggers method that enables forcing value of input *)
	bResetForceValue		: BOOL;				(* Triggers method that enables forcing value of input *)
	
	nFallingTriggerCounter	: USINT;			(* Falling trigger count *)
	nRisingTriggerCounter	: USINT;			(* Rising trigger count *)
	
	piTestSensor 			: FB_DigitalInput;	(* Digital input object *)
END_VAR

IF bFirstCycle THEN
	bFirstCycle := FALSE;
	piTestSensor.MR_FirstCycle('My test digital input');
END_IF

(* Control input simulation *)
piTestSensor.EnableForce := bEnableForce;

(* Assign status variables *)
bValue := piTestSensor.In;
bRisingTrigger := piTestSensor.RisingTrigger;
bFallingTrigger := piTestSensor.FallingTrigger;

(* Count falling trigger *)
IF bFallingTrigger THEN
	nFallingTriggerCounter := nFallingTriggerCounter + 1;
END_IF

(* Count rising trigger *)
IF bRisingTrigger THEN
	nRisingTriggerCounter := nRisingTriggerCounter + 1;
END_IF

(* If simulation of input enabled set it's value to TRUE *)
IF bSetForceValue THEN
	bSetForceValue := FALSE;
	piTestSensor.MR_SetForceValue();
END_IF

(* If simulation of input enabled set it's value to FALSE *)
IF bResetForceValue THEN
	bResetForceValue := FALSE;
	piTestSensor.MR_ResetForceValue();
END_IF

piTestSensor();

END_PROGRAM

// ---- POUs/Universal Blocks/Digital Devices/Digital Input/PRG_FB_DigitalInputExt_Test.TcPOU
PROGRAM PRG_FB_DigitalInputExt_Test
VAR
	bFirstCycle : BOOL := TRUE;
	
	bIn						: BOOL;					(* Current value of input from object *)
	bEnableForce			: BOOL;					(* Enables forcing in digital input object *)
	bFallingTrigger			: BOOL;					(* Falling trigger detected bit *)
	bRisingTrigger			: BOOL;					(* Rising trigger detected bit *)
	bSetForceValue			: BOOL;					(* Triggers method that enables forcing value of input *)
	bResetForceValue		: BOOL;					(* Triggers method that enables forcing value of input *)
	
	nFallingTriggerCounter	: USINT;				(* Falling trigger count *)
	nRisingTriggerCounter	: USINT;				(* Rising trigger count *)
	
	piTestSensor 			: FB_DigitalInputExt;	(* Extended digital input object *)
	
	bInit					: BOOL;
	bAbort  				: BOOL;
	bReset 					: BOOL;
	bStartTracking			: BOOL;
	
	iState					: USINT;
	bActive					: BOOL;
	bErrorTimedout			: BOOL;
	CurrentTimeout			: TIME;
END_VAR

IF bFirstCycle THEN
	bFirstCycle := FALSE;
	piTestSensor.MR_FirstCycleEx( 	sName := 'Test_Sensor',
									bEnableTimeout := TRUE,
									tDefaultTimeout := T#10S);
END_IF

(* Control input simulation *)
piTestSensor.EnableForce := bEnableForce;

(* Assign status variables *)
bIn := piTestSensor.In;
bRisingTrigger := piTestSensor.RisingTrigger;
bFallingTrigger := piTestSensor.FallingTrigger;

(* Count falling trigger *)
IF bFallingTrigger THEN
	nFallingTriggerCounter := nFallingTriggerCounter + 1;
END_IF

(* Count rising trigger *)
IF bRisingTrigger THEN
	nRisingTriggerCounter := nRisingTriggerCounter + 1;
END_IF

(* If simulation of input enabled set it's value to TRUE *)
IF bSetForceValue THEN
	bSetForceValue := FALSE;
	piTestSensor.MR_SetForceValue();
END_IF

